  MoveL 3296 to (-321.69, 3.65, -16.53) mm, rotated rx -179.9 ry 0 rz -90 deg; joints [12.696, -89.548, 135.077, -162.211, 45.978, 167.852]
  MoveL 3297 to (-322.96, 3.57, -14.75) mm, rotated rx -179.9 ry 0 rz -90 deg; joints [12.649, -89.681, 135.215, -162.276, 45.973, 167.898]
  MoveL 3298 to (-323.52, 3.49, -12.64) mm, rotated rx -179.9 ry 0 rz -90 deg; joints [12.644, -89.825, 135.365, -162.283, 45.976, 167.904]
  MoveL 3299 to (-323.29, 3.42, -10.47) mm, rotated rx -179.9 ry 0 rz -90 deg; joints [12.684, -89.963, 135.506, -162.231, 45.988, 167.869]
  MoveL 3300 to (-322.29, 3.34, -8.52) mm, rotated rx -179.9 ry 0 rz -90 deg; joints [12.762, -90.074, 135.62, -162.126, 46.008, 167.798]
  MoveL 3301 to (-320.67, 3.26, -7.05) mm, rotated rx -179.9 ry 0 rz -90 deg; joints [12.868, -90.144, 135.694, -161.983, 46.035, 167.701]
  MoveL 3302 to (-318.64, 3.19, -6.26) mm, rotated rx -179.9 ry 0 rz -90 deg; joints [12.989, -90.162, 135.717, -161.82, 46.066, 167.592]
  MoveL 3303 to (-316.45, 3.11, -6.24) mm, rotated rx -179.9 ry 0 rz -90 deg; joints [13.109, -90.127, 135.687, -161.661, 46.097, 167.484]
  MoveL 3304 to (-314.4, 3.03, -7.01) mm, rotated rx -179.9 ry 0 rz -90 deg; joints [13.21, -90.041, 135.609, -161.525, 46.126, 167.394]
  MoveL 3305 to (-312.76, 2.96, -8.46) mm, rotated rx -179.9 ry 0 rz -90 deg; joints [13.28, -89.916, 135.492, -161.433, 46.15, 167.332]
  MoveL 3306 to (-311.74, 2.88, -10.39) mm, rotated rx -179.9 ry 0 rz -90 deg; joints [13.311, -89.769, 135.353, -161.394, 46.164, 167.308]
  MoveL 3307 to (-311.48, 2.8, -12.56) mm, rotated rx -179.9 ry 0 rz -90 deg; joints [13.297, -89.617, 135.21, -161.416, 46.169, 167.325]
  MoveL 3308 to (-312.01, 2.73, -14.68) mm, rotated rx -179.9 ry 0 rz -90 deg; joints [13.241, -89.482, 135.083, -161.493, 46.165, 167.38]
  MoveL 3309 to (-313.26, 2.65, -16.48) mm, rotated rx -179.9 ry 0 rz -90 deg; joints [13.151, -89.379, 134.988, -161.618, 46.152, 167.466]
  MoveL 3310 to (-315.07, 2.57, -17.71) mm, rotated rx -179.9 ry 0 rz -90 deg; joints [13.038, -89.322, 134.939, -161.773, 46.135, 167.573]
  MoveL 3311 to (-317.2, 2.5, -18.21) mm, rotated rx -179.9 ry 0 rz -90 deg; joints [12.918, -89.317, 134.941, -161.938, 46.116, 167.688]
  MoveL 3312 to (-319.37, 2.42, -17.92) mm, rotated rx -179.9 ry 0 rz -90 deg; joints [12.804, -89.364, 134.996, -162.094, 46.099, 167.796]
  MoveL 3313 to (-321.29, 2.34, -16.88) mm, rotated rx -179.9 ry 0 rz -90 deg; joints [12.714, -89.458, 135.097, -162.219, 46.086, 167.883]
  MoveL 3314 to (-322.71, 2.27, -15.22) mm, rotated rx -179.9 ry 0 rz -90 deg; joints [12.657, -89.585, 135.23, -162.298, 46.079, 167.937]
  MoveL 3315 to (-323.46, 2.19, -13.17) mm, rotated rx -179.9 ry 0 rz -90 deg; joints [12.642, -89.728, 135.378, -162.319, 46.081, 167.953]
  MoveL 3316 to (-323.42, 2.11, -10.98) mm, rotated rx -179.9 ry 0 rz -90 deg; joints [12.671, -89.869, 135.523, -162.281, 46.091, 167.928]
  MoveL 3317 to (-322.6, 2.04, -8.95) mm, rotated rx -179.9 ry 0 rz -90 deg; joints [12.741, -89.988, 135.646, -162.188, 46.109, 167.866]
  MoveL 3318 to (-321.11, 1.96, -7.35) mm, rotated rx -179.9 ry 0 rz -90 deg; joints [12.841, -90.069, 135.73, -162.052, 46.135, 167.774]
  MoveL 3319 to (-319.15, 1.88, -6.38) mm, rotated rx -179.9 ry 0 rz -90 deg; joints [12.96, -90.1, 135.766, -161.893, 46.165, 167.666]
  MoveL 3320 to (-316.98, 1.81, -6.18) mm, rotated rx -179.9 ry 0 rz -90 deg; joints [13.081, -90.077, 135.749, -161.731, 46.196, 167.557]
  MoveL 3321 to (-314.87, 1.73, -6.76) mm, rotated rx -179.9 ry 0 rz -90 deg; joints [13.188, -90.003, 135.681, -161.588, 46.226, 167.462]
  MoveL 3322 to (-313.11, 1.65, -8.05) mm, rotated rx -179.9 ry 0 rz -90 deg; joints [13.267, -89.886, 135.572, -161.484, 46.251, 167.393]
  MoveL 3323 to (-311.92, 1.57, -9.89) mm, rotated rx -179.9 ry 0 rz -90 deg; joints [13.308, -89.743, 135.437, -161.432, 46.268, 167.359]
  MoveL 3324 to (-311.47, 1.5, -12.03) mm, rotated rx -179.9 ry 0 rz -90 deg; joints [13.305, -89.591, 135.293, -161.438, 46.275, 167.366]
  MoveL 3325 to (-311.81, 1.42, -14.19) mm, rotated rx -179.9 ry 0 rz -90 deg; joints [13.259, -89.45, 135.16, -161.503, 46.272, 167.412]
  MoveL 3326 to (-312.9, 1.34, -16.09) mm, rotated rx -179.9 ry 0 rz -90 deg; joints [13.176, -89.338, 135.056, -161.617, 46.261, 167.491]
  MoveL 3327 to (-314.6, 1.27, -17.47) mm, rotated rx -179.9 ry 0 rz -90 deg; joints [13.067, -89.269, 134.995, -161.766, 46.245, 167.594]
  MoveL 3328 to (-316.67, 1.19, -18.16) mm, rotated rx -179.9 ry 0 rz -90 deg; joints [12.947, -89.251, 134.985, -161.931, 46.226, 167.708]
  MoveL 3329 to (-318.86, 1.11, -18.06) mm, rotated rx -179.9 ry 0 rz -90 deg; joints [12.831, -89.286, 135.028, -162.09, 46.208, 167.818]
  MoveL 3330 to (-320.86, 1.04, -17.2) mm, rotated rx -179.9 ry 0 rz -90 deg; joints [12.733, -89.369, 135.118, -162.224, 46.194, 167.911]
  MoveL 3331 to (-322.43, 0.96, -15.67) mm, rotated rx -179.9 ry 0 rz -90 deg; joints [12.667, -89.49, 135.244, -162.315, 46.187, 167.974]
  MoveL 3332 to (-323.35, 0.88, -13.69) mm, rotated rx -179.9 ry 0 rz -90 deg; joints [12.642, -89.631, 135.391, -162.351, 46.186, 168]
  MoveL 3333 to (-323.5, 0.81, -11.5) mm, rotated rx -179.9 ry 0 rz -90 deg; joints [12.661, -89.774, 135.539, -162.328, 46.195, 167.985]
  MoveL 3334 to (-322.86, 0.73, -9.41) mm, rotated rx -179.9 ry 0 rz -90 deg; joints [12.721, -89.9, 135.668, -162.247, 46.211, 167.931]
  MoveL 3335 to (-321.52, 0.65, -7.69) mm, rotated rx -179.9 ry 0 rz -90 deg; joints [12.815, -89.991, 135.763, -162.12, 46.235, 167.845]
  MoveL 3336 to (-319.65, 0.58, -6.55) mm, rotated rx -179.9 ry 0 rz -90 deg; joints [12.931, -90.035, 135.812, -161.965, 46.264, 167.741]
  MoveL 3337 to (-317.5, 0.5, -6.15) mm, rotated rx -179.9 ry 0 rz -90 deg; joints [13.053, -90.025, 135.807, -161.802, 46.295, 167.631]
  MoveL 3338 to (-317.17, 0.5, -6.15) mm, rotated rx -179.9 ry 0 rz -90 deg; joints [13.071, -90.02, 135.802, -161.777, 46.299, 167.614]
  MoveC 3339 to (-315.68, 0.5, -6.77) mm, rotated rx -179.9 ry 0 rz -90 deg; joints [13.145, -89.956, 135.739, -161.678, 46.316, 167.547] to (-315.06, 0.5, -8.27) mm, rotated rx -179.9 ry 0 rz -90 deg; joints [13.159, -89.848, 135.632, -161.659, 46.32, 167.535]
  MoveL 3340 to (-315.06, 0.5, -8.27) mm, rotated rx -179.9 ry 0 rz -90 deg; joints [13.159, -89.848, 135.632, -161.659, 46.32, 167.535]
  MoveL 3341 to (-315.06, 0.5, -303.97) mm, rotated rx -179.9 ry 0 rz -90 deg; joints [10.211, -71.759, 114.391, -164.852, 42.693, 169.127]
  MoveC 3342 to (-315.68, 0.5, -305.46) mm, rotated rx -179.9 ry 0 rz -90 deg; joints [10.173, -71.679, 114.282, -164.899, 42.658, 169.156] to (-317.17, 0.5, -306.08) mm, rotated rx -179.9 ry 0 rz -90 deg; joints [10.104, -71.658, 114.254, -164.997, 42.639, 169.225]
  MoveL 3343 to (-317.17, 0.5, -306.08) mm, rotated rx -179.9 ry 0 rz -90 deg; joints [10.104, -71.658, 114.254, -164.997, 42.639, 169.225]
  MoveL 3344 to (-317.84, 0.5, -306.08) mm, rotated rx -179.9 ry 0 rz -90 deg; joints [10.076, -71.665, 114.264, -165.039, 42.636, 169.256]
  MoveC 3345 to (-319.33, 0.5, -305.46) mm, rotated rx -179.9 ry 0 rz -90 deg; joints [10.016, -71.716, 114.334, -165.13, 42.643, 169.326] to (-319.95, 0.5, -303.97) mm, rotated rx -179.9 ry 0 rz -90 deg; joints [10.001, -71.809, 114.461, -165.161, 42.673, 169.354]
  MoveL 3346 to (-319.95, 0.5, -303.97) mm, rotated rx -179.9 ry 0 rz -90 deg; joints [10.001, -71.809, 114.461, -165.161, 42.673, 169.354]
  MoveL 3347 to (-319.95, 0.5, -8.27) mm, rotated rx -179.9 ry 0 rz -90 deg; joints [12.894, -89.922, 135.707, -162.018, 46.264, 167.779]
  MoveC 3348 to (-319.33, 0.5, -6.77) mm, rotated rx -179.9 ry 0 rz -90 deg; joints [12.946, -90.012, 135.795, -161.947, 46.273, 167.73] to (-317.84, 0.5, -6.15) mm, rotated rx -179.9 ry 0 rz -90 deg; joints [13.035, -90.03, 135.812, -161.826, 46.292, 167.648]
  MoveL 3349 to (-317.84, 0.5, -6.15) mm, rotated rx -179.9 ry 0 rz -90 deg; joints [13.035, -90.03, 135.812, -161.826, 46.292, 167.648]
  MoveL 3350 to (-317.5, 0.5, -6.15) mm, rotated rx -179.9 ry 0 rz -90 deg; joints [13.053, -90.025, 135.807, -161.802, 46.295, 167.631]
  MoveC 3351 to (-315.43, 0.5, -5.57) mm, rotated rx -179.9 ry 0 rz -90 deg; joints [13.174, -90.032, 135.813, -161.639, 46.32, 167.52] to (-313.95, 0.5, -4) mm, rotated rx -179.9 ry 0 rz -90 deg; joints [13.275, -90.114, 135.892, -161.502, 46.34, 167.427]
  MoveL 3352 to (-313.95, 0.5, -4) mm, rotated rx -179.9 ry 0 rz -90 deg; joints [13.275, -90.114, 135.892, -161.502, 46.34, 167.427]
  MoveC 3353 to (-311.54, 0.5, -2.91) mm, rotated rx -179.9 ry 0 rz -90 deg; joints [13.42, -90.149, 135.924, -161.306, 46.37, 167.293] to (-309.91, 0.5, -4.99) mm, rotated rx -179.9 ry 0 rz -90 deg; joints [13.481, -89.985, 135.763, -161.224, 46.386, 167.238]
  MoveL 3354 to (-309.91, 0.5, -4.99) mm, rotated rx -179.9 ry 0 rz -90 deg; joints [13.481, -89.985, 135.763, -161.224, 46.386, 167.238]
  MoveL 3355 to (-309.91, 0.5, -311.23) mm, rotated rx -179.9 ry 0 rz -90 deg; joints [10.374, -71.283, 113.739, -164.566, 42.556, 168.888]
  MoveL 3356 to (-325.1, 0.5, -311.23) mm, rotated rx -179.9 ry 0 rz -90 deg; joints [9.727, -71.437, 113.959, -165.524, 42.495, 169.594]
  MoveL 3357 to (-325.1, 0.5, -1) mm, rotated rx -179.9 ry 0 rz -90 deg; joints [12.703, -90.482, 136.257, -162.273, 46.213, 167.95]
  MoveL 3358 to (-309.91, 0.5, -1) mm, rotated rx -179.9 ry 0 rz -90 deg; joints [13.534, -90.25, 136.022, -161.151, 46.392, 167.188]
  MoveL 3359 to (-309.91, 0.5, -4.99) mm, rotated rx -179.9 ry 0 rz -90 deg; joints [13.481, -89.985, 135.763, -161.224, 46.386, 167.238]
  MoveL 3360 to (-309.93, 0.52, -5.21) mm, rotated rx -179.9 ry 0 rz -90 deg; joints [13.477, -89.972, 135.749, -161.229, 46.384, 167.241]
  MoveL 3361 to (-309.98, 0.58, -5.42) mm, rotated rx -179.9 ry 0 rz -90 deg; joints [13.472, -89.962, 135.734, -161.235, 46.379, 167.244]
  MoveL 3362 to (-310.06, 0.67, -5.6) mm, rotated rx -179.9 ry 0 rz -90 deg; joints [13.465, -89.955, 135.72, -161.242, 46.37, 167.247]
  MoveL 3363 to (-310.16, 0.8, -5.75) mm, rotated rx -179.9 ry 0 rz -90 deg; joints [13.457, -89.953, 135.707, -161.249, 46.358, 167.249]
  MoveL 3364 to (-310.26, 0.95, -5.87) mm, rotated rx -179.9 ry 0 rz -90 deg; joints [13.45, -89.954, 135.695, -161.254, 46.344, 167.25]
  MoveL 3365 to (-310.36, 1.13, -5.96) mm, rotated rx -179.9 ry 0 rz -90 deg; joints [13.444, -89.958, 135.684, -161.258, 46.328, 167.249]
  MoveL 3366 to (-310.43, 1.34, -6.02) mm, rotated rx -179.9 ry 0 rz -90 deg; joints [13.439, -89.965, 135.674, -161.259, 46.311, 167.246]
  MoveL 3367 to (-310.48, 1.55, -6.05) mm, rotated rx -179.9 ry 0 rz -90 deg; joints [13.436, -89.974, 135.665, -161.258, 46.293, 167.241]
  MoveL 3368 to (-310.49, 1.77, -6.06) mm, rotated rx -179.9 ry 0 rz -90 deg; joints [13.435, -89.984, 135.656, -161.254, 46.276, 167.233]
  Set speed (1000.0 mm/s)
  MoveL 3369 to (-310.49, 185.53, -6.06) mm, rotated rx -179.9 ry 0 rz -90 deg; joints [13.36, -96.669, 127.503, -154.519, 32.472, 158.531]
  Print: /'Contour3'
  Call SetTool(1)
  Set speed (1000.0 mm/s)
  MoveL 3370 to (-315.03, 25.52, 4.01) mm, rotated rx -179.9 ry 0 rz -90 deg; joints [13.309, -91.824, 135.461, -160.771, 44.323, 166.421]
  MoveL 3371 to (-315.03, 11.79, 4.01) mm, rotated rx -179.9 ry 0 rz -90 deg; joints [13.315, -91.197, 135.998, -161.144, 45.423, 166.953]
  Set speed (100.0 mm/s)
  MoveL 3372 to (-315.03, 4.8, 4.01) mm, rotated rx -179.9 ry 0 rz -90 deg; joints [13.318, -90.869, 136.265, -161.327, 45.987, 167.218]
  MoveL 3373 to (-314.68, 3.9, 3.89) mm, rotated rx -179.9 ry 0 rz -90 deg; joints [13.336, -90.813, 136.286, -161.326, 46.064, 167.236]
  MoveL 3374 to (-313.82, 3.52, 3.62) mm, rotated rx -179.9 ry 0 rz -90 deg; joints [13.38, -90.764, 136.269, -161.277, 46.105, 167.21]
  MoveL 3375 to (-309.98, 3.52, 2.4) mm, rotated rx -179.9 ry 0 rz -90 deg; joints [13.574, -90.622, 136.13, -161.015, 46.151, 167.032]
  MoveC 3376 to (-309.23, 3.53, 1.78) mm, rotated rx -179.9 ry 0 rz -90 deg; joints [13.606, -90.568, 136.077, -160.972, 46.16, 167.003] to (-309.15, 3.53, 0.81) mm, rotated rx -179.9 ry 0 rz -90 deg; joints [13.598, -90.502, 136.014, -160.984, 46.16, 167.012]
  MoveL 3377 to (-309.15, 3.52, 0.81) mm, rotated rx -179.9 ry 0 rz -90 deg; joints [13.598, -90.502, 136.014, -160.984, 46.16, 167.012]
  MoveL 3378 to (-309.24, 3.53, 0.47) mm, rotated rx -179.9 ry 0 rz -90 deg; joints [13.588, -90.481, 135.993, -160.997, 46.159, 167.021]
  MoveL 3379 to (-309.31, 3.52, 0.13) mm, rotated rx -179.9 ry 0 rz -90 deg; joints [13.58, -90.46, 135.972, -161.009, 46.157, 167.029]
  MoveL 3380 to (-309.38, 3.52, -0.32) mm, rotated rx -179.9 ry 0 rz -90 deg; joints [13.57, -90.431, 135.944, -161.022, 46.156, 167.038]
  MoveL 3381 to (-309.41, 3.52, -0.77) mm, rotated rx -179.9 ry 0 rz -90 deg; joints [13.563, -90.401, 135.916, -161.032, 46.155, 167.045]
  MoveL 3382 to (-309.41, 3.52, -1.67) mm, rotated rx -179.9 ry 0 rz -90 deg; joints [13.551, -90.342, 135.858, -161.049, 46.154, 167.057]
  MoveL 3383 to (-309.41, 3.53, -310.57) mm, rotated rx -179.9 ry 0 rz -90 deg; joints [10.399, -71.426, 113.69, -164.473, 42.376, 168.785]
  MoveL 3384 to (-309.41, 3.52, -311.47) mm, rotated rx -179.9 ry 0 rz -90 deg; joints [10.392, -71.373, 113.619, -164.478, 42.356, 168.785]
  MoveL 3385 to (-309.38, 3.52, -311.92) mm, rotated rx -179.9 ry 0 rz -90 deg; joints [10.39, -71.347, 113.583, -164.478, 42.347, 168.783]
  MoveL 3386 to (-309.31, 3.52, -312.37) mm, rotated rx -179.9 ry 0 rz -90 deg; joints [10.389, -71.32, 113.546, -164.476, 42.337, 168.78]
  MoveL 3387 to (-309.24, 3.52, -312.7) mm, rotated rx -179.9 ry 0 rz -90 deg; joints [10.39, -71.299, 113.518, -164.474, 42.33, 168.777]
  MoveL 3388 to (-309.15, 3.53, -313.04) mm, rotated rx -179.9 ry 0 rz -90 deg; joints [10.391, -71.279, 113.49, -164.47, 42.323, 168.773]
  MoveL 3389 to (-309.08, 3.53, -313.26) mm, rotated rx -179.9 ry 0 rz -90 deg; joints [10.392, -71.265, 113.471, -164.466, 42.318, 168.769]
  MoveL 3390 to (-308.91, 3.52, -313.71) mm, rotated rx -179.9 ry 0 rz -90 deg; joints [10.396, -71.237, 113.433, -164.458, 42.309, 168.761]
  MoveL 3391 to (-308.7, 3.52, -314.16) mm, rotated rx -179.9 ry 0 rz -90 deg; joints [10.401, -71.209, 113.394, -164.447, 42.3, 168.751]
  MoveL 3392 to (-308.49, 3.53, -314.53) mm, rotated rx -179.9 ry 0 rz -90 deg; joints [10.407, -71.185, 113.362, -164.436, 42.293, 168.742]
  MoveL 3393 to (-308.25, 3.53, -314.9) mm, rotated rx -179.9 ry 0 rz -90 deg; joints [10.414, -71.161, 113.329, -164.423, 42.286, 168.73]
  MoveL 3394 to (-308.13, 3.52, -315.06) mm, rotated rx -179.9 ry 0 rz -90 deg; joints [10.418, -71.15, 113.314, -164.416, 42.283, 168.725]
  MoveL 3395 to (-307.96, 3.53, -315.27) mm, rotated rx -179.9 ry 0 rz -90 deg; joints [10.424, -71.136, 113.295, -164.406, 42.278, 168.717]
  MoveL 3396 to (-307.78, 3.53, -315.49) mm, rotated rx -179.9 ry 0 rz -90 deg; joints [10.43, -71.122, 113.275, -164.396, 42.274, 168.708]
  MoveL 3397 to (-307.57, 3.52, -315.7) mm, rotated rx -179.9 ry 0 rz -90 deg; joints [10.437, -71.107, 113.255, -164.384, 42.271, 168.699]
  MoveL 3398 to (-307.35, 3.53, -315.92) mm, rotated rx -179.9 ry 0 rz -90 deg; joints [10.444, -71.092, 113.234, -164.371, 42.267, 168.688]
  MoveL 3399 to (-307.31, 3.52, -315.96) mm, rotated rx -179.9 ry 0 rz -90 deg; joints [10.446, -71.089, 113.23, -164.369, 42.266, 168.686]
  MoveL 3400 to (-306.88, 3.52, -316.31) mm, rotated rx -179.9 ry 0 rz -90 deg; joints [10.461, -71.064, 113.196, -164.343, 42.26, 168.666]
  MoveL 3401 to (-306.45, 3.53, -316.6) mm, rotated rx -179.9 ry 0 rz -90 deg; joints [10.477, -71.043, 113.166, -164.318, 42.255, 168.646]
  MoveL 3402 to (-306.02, 3.53, -316.86) mm, rotated rx -179.9 ry 0 rz -90 deg; joints [10.493, -71.023, 113.139, -164.292, 42.251, 168.626]
  MoveL 3403 to (-305.55, 3.53, -317.08) mm, rotated rx -179.9 ry 0 rz -90 deg; joints [10.511, -71.006, 113.115, -164.264, 42.249, 168.604]
  MoveL 3404 to (-305.1, 3.52, -317.25) mm, rotated rx -179.9 ry 0 rz -90 deg; joints [10.529, -70.991, 113.094, -164.237, 42.247, 168.583]
  MoveL 3405 to (-304.66, 3.53, -317.38) mm, rotated rx -179.9 ry 0 rz -90 deg; joints [10.547, -70.978, 113.077, -164.209, 42.245, 168.562]
  MoveL 3406 to (-304.21, 3.52, -317.48) mm, rotated rx -179.9 ry 0 rz -90 deg; joints [10.565, -70.968, 113.062, -164.181, 42.245, 168.541]
  MoveL 3407 to (-303.76, 3.53, -317.55) mm, rotated rx -179.9 ry 0 rz -90 deg; joints [10.583, -70.959, 113.05, -164.153, 42.246, 168.52]
  MoveL 3408 to (-303.31, 3.52, -317.58) mm, rotated rx -179.9 ry 0 rz -90 deg; joints [10.602, -70.952, 113.04, -164.125, 42.247, 168.499]
  MoveL 3409 to (-302.86, 3.53, -317.59) mm, rotated rx -179.9 ry 0 rz -90 deg; joints [10.621, -70.947, 113.033, -164.097, 42.248, 168.478]
  MoveL 3410 to (315.44, 3.53, -317.59) mm, rotated rx -179.9 ry 0 rz -90 deg; joints [33.379, -56.906, 91.665, -130.07, 45.953, 141.252]
  MoveL 3411 to (315.89, 3.53, -317.58) mm, rotated rx -179.9 ry 0 rz -90 deg; joints [33.393, -56.891, 91.641, -130.048, 45.956, 141.232]
  MoveL 3412 to (316.34, 3.52, -317.54) mm, rotated rx -179.9 ry 0 rz -90 deg; joints [33.407, -56.878, 91.62, -130.026, 45.96, 141.213]
  MoveL 3413 to (316.79, 3.53, -317.47) mm, rotated rx -179.9 ry 0 rz -90 deg; joints [33.422, -56.866, 91.601, -130.004, 45.965, 141.194]
  MoveL 3414 to (317.24, 3.52, -317.36) mm, rotated rx -179.9 ry 0 rz -90 deg; joints [33.438, -56.856, 91.584, -129.983, 45.97, 141.175]
  MoveL 3415 to (317.69, 3.53, -317.23) mm, rotated rx -179.9 ry 0 rz -90 deg; joints [33.454, -56.848, 91.571, -129.961, 45.977, 141.158]
  MoveL 3416 to (318.14, 3.52, -317.05) mm, rotated rx -179.9 ry 0 rz -90 deg; joints [33.472, -56.842, 91.561, -129.939, 45.986, 141.141]
  MoveL 3417 to (318.54, 3.52, -316.86) mm, rotated rx -179.9 ry 0 rz -90 deg; joints [33.488, -56.838, 91.555, -129.92, 45.994, 141.126]
  MoveL 3418 to (318.78, 3.52, -316.72) mm, rotated rx -179.9 ry 0 rz -90 deg; joints [33.498, -56.837, 91.552, -129.908, 46, 141.117]
  MoveL 3419 to (319.03, 3.53, -316.56) mm, rotated rx -179.9 ry 0 rz -90 deg; joints [33.509, -56.836, 91.551, -129.896, 46.006, 141.109]
  MoveL 3420 to (319.43, 3.52, -316.28) mm, rotated rx -179.9 ry 0 rz -90 deg; joints [33.526, -56.837, 91.552, -129.877, 46.018, 141.096]
  MoveL 3421 to (319.83, 3.52, -315.96) mm, rotated rx -179.9 ry 0 rz -90 deg; joints [33.545, -56.841, 91.557, -129.859, 46.03, 141.084]
  MoveL 3422 to (319.93, 3.53, -315.86) mm, rotated rx -179.9 ry 0 rz -90 deg; joints [33.55, -56.842, 91.56, -129.853, 46.034, 141.081]
  MoveL 3423 to (320.14, 3.52, -315.66) mm, rotated rx -179.9 ry 0 rz -90 deg; joints [33.56, -56.846, 91.565, -129.844, 46.042, 141.076]
  MoveL 3424 to (320.32, 3.52, -315.46) mm, rotated rx -179.9 ry 0 rz -90 deg; joints [33.57, -56.85, 91.571, -129.835, 46.049, 141.071]
  MoveL 3425 to (320.65, 3.53, -315.06) mm, rotated rx -179.9 ry 0 rz -90 deg; joints [33.588, -56.859, 91.586, -129.82, 46.064, 141.063]
  MoveL 3426 to (320.83, 3.52, -314.8) mm, rotated rx -179.9 ry 0 rz -90 deg; joints [33.599, -56.866, 91.597, -129.811, 46.073, 141.06]
  MoveL 3427 to (321.04, 3.52, -314.48) mm, rotated rx -179.9 ry 0 rz -90 deg; joints [33.612, -56.876, 91.612, -129.801, 46.085, 141.056]
  MoveL 3428 to (321.22, 3.52, -314.16) mm, rotated rx -179.9 ry 0 rz -90 deg; joints [33.623, -56.887, 91.629, -129.793, 46.096, 141.054]
  MoveL 3429 to (321.43, 3.53, -313.71) mm, rotated rx -179.9 ry 0 rz -90 deg; joints [33.639, -56.903, 91.654, -129.783, 46.112, 141.053]
  MoveL 3430 to (321.6, 3.53, -313.26) mm, rotated rx -179.9 ry 0 rz -90 deg; joints [33.653, -56.92, 91.682, -129.775, 46.127, 141.053]
  MoveL 3431 to (321.73, 3.53, -312.81) mm, rotated rx -179.9 ry 0 rz -90 deg; joints [33.666, -56.939, 91.711, -129.769, 46.143, 141.055]
  MoveL 3432 to (321.83, 3.52, -312.37) mm, rotated rx -179.9 ry 0 rz -90 deg; joints [33.678, -56.959, 91.743, -129.765, 46.158, 141.059]
  MoveL 3433 to (321.89, 3.52, -311.92) mm, rotated rx -179.9 ry 0 rz -90 deg; joints [33.69, -56.98, 91.776, -129.762, 46.173, 141.064]
  MoveL 3434 to (321.93, 3.52, -311.47) mm, rotated rx -179.9 ry 0 rz -90 deg; joints [33.7, -57.002, 91.811, -129.761, 46.187, 141.07]
  MoveL 3435 to (321.93, 3.52, -310.57) mm, rotated rx -179.9 ry 0 rz -90 deg; joints [33.718, -57.049, 91.885, -129.761, 46.216, 141.086]
  MoveL 3436 to (321.93, 3.52, -1.67) mm, rotated rx -179.9 ry 0 rz -90 deg; joints [41.183, -71.832, 113.655, -126.643, 55.135, 143.485]
  MoveL 3437 to (321.93, 3.52, -0.77) mm, rotated rx -179.9 ry 0 rz -90 deg; joints [41.209, -71.873, 113.709, -126.626, 55.158, 143.485]
  MoveL 3438 to (321.89, 3.52, -0.32) mm, rotated rx -179.9 ry 0 rz -90 deg; joints [41.221, -71.894, 113.738, -126.619, 55.17, 143.486]
  MoveL 3439 to (321.83, 3.53, 0.13) mm, rotated rx -179.9 ry 0 rz -90 deg; joints [41.231, -71.917, 113.769, -126.613, 55.181, 143.487]
  MoveL 3440 to (321.73, 3.52, 0.58) mm, rotated rx -179.9 ry 0 rz -90 deg; joints [41.241, -71.941, 113.801, -126.608, 55.192, 143.49]
  MoveL 3441 to (321.6, 3.53, 1.03) mm, rotated rx -179.9 ry 0 rz -90 deg; joints [41.25, -71.966, 113.835, -126.605, 55.202, 143.494]
  MoveL 3442 to (321.43, 3.53, 1.48) mm, rotated rx -179.9 ry 0 rz -90 deg; joints [41.257, -71.993, 113.871, -126.603, 55.212, 143.5]
  MoveL 3443 to (321.22, 3.52, 1.93) mm, rotated rx -179.9 ry 0 rz -90 deg; joints [41.263, -72.021, 113.91, -126.603, 55.221, 143.506]
  MoveL 3444 to (321.04, 3.53, 2.25) mm, rotated rx -179.9 ry 0 rz -90 deg; joints [41.266, -72.042, 113.938, -126.603, 55.228, 143.512]
  MoveL 3445 to (320.83, 3.52, 2.57) mm, rotated rx -179.9 ry 0 rz -90 deg; joints [41.269, -72.065, 113.969, -126.605, 55.234, 143.518]
  MoveL 3446 to (320.65, 3.53, 2.82) mm, rotated rx -179.9 ry 0 rz -90 deg; joints [41.27, -72.083, 113.994, -126.608, 55.239, 143.524]
  MoveL 3447 to (320.32, 3.52, 3.22) mm, rotated rx -179.9 ry 0 rz -90 deg; joints [41.271, -72.114, 114.035, -126.613, 55.246, 143.534]
  MoveL 3448 to (320.14, 3.52, 3.42) mm, rotated rx -179.9 ry 0 rz -90 deg; joints [41.271, -72.13, 114.057, -126.617, 55.249, 143.54]
  MoveL 3449 to (319.93, 3.52, 3.62) mm, rotated rx -179.9 ry 0 rz -90 deg; joints [41.27, -72.147, 114.08, -126.621, 55.252, 143.546]
  MoveL 3450 to (319.83, 3.53, 3.72) mm, rotated rx -179.9 ry 0 rz -90 deg; joints [41.269, -72.156, 114.092, -126.623, 55.254, 143.55]
  MoveL 3451 to (319.43, 3.53, 4.05) mm, rotated rx -179.9 ry 0 rz -90 deg; joints [41.266, -72.186, 114.133, -126.633, 55.258, 143.562]
  MoveL 3452 to (319.03, 3.52, 4.33) mm, rotated rx -179.9 ry 0 rz -90 deg; joints [41.261, -72.214, 114.171, -126.643, 55.261, 143.574]
  MoveL 3453 to (318.79, 3.53, 4.48) mm, rotated rx -179.9 ry 0 rz -90 deg; joints [41.257, -72.23, 114.193, -126.65, 55.262, 143.582]
  MoveL 3454 to (318.54, 3.53, 4.62) mm, rotated rx -179.9 ry 0 rz -90 deg; joints [41.253, -72.246, 114.215, -126.657, 55.263, 143.59]
  MoveL 3455 to (318.14, 3.52, 4.81) mm, rotated rx -179.9 ry 0 rz -90 deg; joints [41.245, -72.27, 114.248, -126.669, 55.264, 143.603]
  MoveL 3456 to (317.69, 3.52, 4.99) mm, rotated rx -179.9 ry 0 rz -90 deg; joints [41.236, -72.296, 114.282, -126.684, 55.264, 143.617]
  MoveL 3457 to (317.24, 3.52, 5.13) mm, rotated rx -179.9 ry 0 rz -90 deg; joints [41.225, -72.319, 114.315, -126.699, 55.263, 143.631]
  MoveL 3458 to (316.79, 3.52, 5.23) mm, rotated rx -179.9 ry 0 rz -90 deg; joints [41.213, -72.342, 114.345, -126.715, 55.26, 143.645]
  MoveL 3459 to (316.34, 3.52, 5.3) mm, rotated rx -179.9 ry 0 rz -90 deg; joints [41.201, -72.362, 114.373, -126.732, 55.257, 143.659]
  MoveL 3460 to (315.89, 3.53, 5.34) mm, rotated rx -179.9 ry 0 rz -90 deg; joints [41.187, -72.381, 114.399, -126.749, 55.254, 143.674]
  MoveL 3461 to (315.44, 3.52, 5.35) mm, rotated rx -179.9 ry 0 rz -90 deg; joints [41.172, -72.399, 114.424, -126.767, 55.249, 143.688]
  MoveL 3462 to (-302.86, 3.52, 5.35) mm, rotated rx -179.9 ry 0 rz -90 deg; joints [14.002, -90.704, 136.204, -160.435, 46.243, 166.636]
  MoveL 3463 to (-303.31, 3.52, 5.35) mm, rotated rx -179.9 ry 0 rz -90 deg; joints [13.978, -90.711, 136.211, -160.468, 46.238, 166.659]
  MoveL 3464 to (-303.76, 3.52, 5.31) mm, rotated rx -179.9 ry 0 rz -90 deg; joints [13.953, -90.716, 136.216, -160.502, 46.232, 166.682]
  MoveL 3465 to (-304.21, 3.52, 5.25) mm, rotated rx -179.9 ry 0 rz -90 deg; joints [13.927, -90.719, 136.22, -160.536, 46.226, 166.705]
  MoveL 3466 to (-304.66, 3.53, 5.15) mm, rotated rx -179.9 ry 0 rz -90 deg; joints [13.901, -90.72, 136.22, -160.571, 46.22, 166.729]
  MoveL 3467 to (-305.1, 3.53, 5.01) mm, rotated rx -179.9 ry 0 rz -90 deg; joints [13.875, -90.718, 136.219, -160.607, 46.215, 166.753]
  MoveL 3468 to (-305.55, 3.53, 4.84) mm, rotated rx -179.9 ry 0 rz -90 deg; joints [13.848, -90.714, 136.215, -160.643, 46.209, 166.778]
  MoveL 3469 to (-306.02, 3.53, 4.62) mm, rotated rx -179.9 ry 0 rz -90 deg; joints [13.82, -90.706, 136.209, -160.682, 46.203, 166.804]
  MoveL 3470 to (-306.45, 3.52, 4.37) mm, rotated rx -179.9 ry 0 rz -90 deg; joints [13.793, -90.697, 136.2, -160.719, 46.197, 166.829]
  MoveL 3471 to (-306.88, 3.53, 4.07) mm, rotated rx -179.9 ry 0 rz -90 deg; joints [13.765, -90.684, 136.188, -160.756, 46.191, 166.855]
  MoveL 3472 to (-307.31, 3.52, 3.72) mm, rotated rx -179.9 ry 0 rz -90 deg; joints [13.737, -90.667, 136.172, -160.794, 46.186, 166.881]
  MoveL 3473 to (-307.35, 3.53, 3.68) mm, rotated rx -179.9 ry 0 rz -90 deg; joints [13.734, -90.665, 136.17, -160.798, 46.185, 166.884]
  MoveL 3474 to (-307.57, 3.53, 3.47) mm, rotated rx -179.9 ry 0 rz -90 deg; joints [13.719, -90.655, 136.16, -160.818, 46.182, 166.898]
  MoveL 3475 to (-307.78, 3.53, 3.25) mm, rotated rx -179.9 ry 0 rz -90 deg; joints [13.705, -90.644, 136.149, -160.837, 46.179, 166.911]
  MoveL 3476 to (-307.96, 3.53, 3.04) mm, rotated rx -179.9 ry 0 rz -90 deg; joints [13.692, -90.632, 136.138, -160.855, 46.177, 166.923]
  MoveL 3477 to (-308.13, 3.53, 2.82) mm, rotated rx -179.9 ry 0 rz -90 deg; joints [13.68, -90.621, 136.127, -160.871, 46.175, 166.934]
  MoveL 3478 to (-308.25, 3.53, 2.66) mm, rotated rx -179.9 ry 0 rz -90 deg; joints [13.672, -90.612, 136.119, -160.883, 46.173, 166.942]
  MoveL 3479 to (-308.49, 3.52, 2.29) mm, rotated rx -179.9 ry 0 rz -90 deg; joints [13.653, -90.591, 136.099, -160.908, 46.17, 166.959]
  MoveL 3480 to (-308.7, 3.52, 1.93) mm, rotated rx -179.9 ry 0 rz -90 deg; joints [13.637, -90.57, 136.078, -160.93, 46.167, 166.974]
  MoveL 3481 to (-308.91, 3.52, 1.48) mm, rotated rx -179.9 ry 0 rz -90 deg; joints [13.62, -90.543, 136.053, -160.954, 46.164, 166.991]
  MoveL 3482 to (-309.08, 3.53, 1.03) mm, rotated rx -179.9 ry 0 rz -90 deg; joints [13.605, -90.516, 136.027, -160.975, 46.161, 167.005]
  MoveL 3483 to (-309.15, 3.52, 0.81) mm, rotated rx -179.9 ry 0 rz -90 deg; joints [13.598, -90.502, 136.014, -160.984, 46.16, 167.012]
  MoveC 3484 to (-309.77, 3.53, 0.07) mm, rotated rx -179.9 ry 0 rz -90 deg; joints [13.554, -90.463, 135.976, -161.044, 46.152, 167.053] to (-310.74, 3.52, -0.02) mm, rotated rx -179.9 ry 0 rz -90 deg; joints [13.5, -90.472, 135.986, -161.117, 46.14, 167.103]
  MoveL 3485 to (-310.74, 3.53, -0.02) mm, rotated rx -179.9 ry 0 rz -90 deg; joints [13.5, -90.472, 135.986, -161.117, 46.14, 167.103]
  MoveC 3486 to (-311.92, 3.53, -0.24) mm, rotated rx -179.9 ry 0 rz -90 deg; joints [13.433, -90.476, 135.99, -161.208, 46.125, 167.165] to (-312.39, 3.52, -1.34) mm, rotated rx -179.9 ry 0 rz -90 deg; joints [13.393, -90.41, 135.926, -161.263, 46.118, 167.203]
  MoveL 3487 to (-312.39, 3.52, -1.34) mm, rotated rx -179.9 ry 0 rz -90 deg; joints [13.393, -90.41, 135.926, -161.263, 46.118, 167.203]
  MoveC 3488 to (-312.56, 3.53, -2.1) mm, rotated rx -179.9 ry 0 rz -90 deg; joints [13.373, -90.362, 135.88, -161.289, 46.115, 167.221] to (-313.14, 3.53, -2.61) mm, rotated rx -179.9 ry 0 rz -90 deg; joints [13.335, -90.337, 135.856, -161.341, 46.108, 167.257]
  MoveL 3489 to (-313.14, 3.52, -2.61) mm, rotated rx -179.9 ry 0 rz -90 deg; joints [13.335, -90.337, 135.856, -161.341, 46.108, 167.257]
  MoveC 3490 to (-321.1, 3.53, 0.46) mm, rotated rx -179.9 ry 0 rz -90 deg; joints [12.94, -90.664, 136.178, -161.875, 46.015, 167.62] to (-318.03, 3.52, 8.42) mm, rotated rx -179.9 ry 0 rz -90 deg; joints [13.211, -91.152, 136.644, -161.501, 46.054, 167.359]
  MoveL 3491 to (-318.03, 3.52, 8.42) mm, rotated rx -179.9 ry 0 rz -90 deg; joints [13.211, -91.152, 136.644, -161.501, 46.054, 167.359]
  MoveC 3492 to (-310.52, 3.52, 6.18) mm, rotated rx -179.9 ry 0 rz -90 deg; joints [13.594, -90.883, 136.382, -160.985, 46.147, 167.009] to (-311.55, 3.52, -1.58) mm, rotated rx -179.9 ry 0 rz -90 deg; joints [13.435, -90.381, 135.897, -161.205, 46.128, 167.164]
  MoveL 3493 to (-311.55, 3.53, -1.58) mm, rotated rx -179.9 ry 0 rz -90 deg; joints [13.435, -90.381, 135.897, -161.205, 46.128, 167.164]
  MoveL 3494 to (-311.58, 3.52, -1.61) mm, rotated rx -179.9 ry 0 rz -90 deg; joints [13.433, -90.379, 135.896, -161.208, 46.128, 167.166]
  MoveL 3495 to (-313.45, 3.45, -2.74) mm, rotated rx -179.9 ry 0 rz -90 deg; joints [13.317, -90.33, 135.855, -161.368, 46.11, 167.277]
  MoveL 3496 to (-315.6, 3.37, -3.13) mm, rotated rx -179.9 ry 0 rz -90 deg; joints [13.195, -90.333, 135.866, -161.536, 46.09, 167.393]
  MoveL 3497 to (-317.75, 3.29, -2.73) mm, rotated rx -179.9 ry 0 rz -90 deg; joints [13.083, -90.389, 135.928, -161.689, 46.071, 167.499]
  MoveL 3498 to (-319.61, 3.22, -1.59) mm, rotated rx -179.9 ry 0 rz -90 deg; joints [12.996, -90.49, 136.034, -161.809, 46.056, 167.581]
  MoveL 3499 to (-320.94, 3.14, 0.13) mm, rotated rx -179.9 ry 0 rz -90 deg; joints [12.944, -90.622, 136.169, -161.879, 46.048, 167.63]
  MoveL 3500 to (-321.58, 3.06, 2.22) mm, rotated rx -179.9 ry 0 rz -90 deg; joints [12.936, -90.768, 136.316, -161.891, 46.048, 167.638]
  MoveL 3501 to (-321.43, 2.99, 4.4) mm, rotated rx -179.9 ry 0 rz -90 deg; joints [12.972, -90.908, 136.457, -161.842, 46.056, 167.605]
  MoveL 3502 to (-320.51, 2.91, 6.38) mm, rotated rx -179.9 ry 0 rz -90 deg; joints [13.048, -91.024, 136.574, -161.74, 46.074, 167.536]
  MoveL 3503 to (-318.96, 2.83, 7.91) mm, rotated rx -179.9 ry 0 rz -90 deg; joints [13.153, -91.099, 136.651, -161.597, 46.099, 167.439]
  MoveL 3504 to (-316.95, 2.76, 8.78) mm, rotated rx -179.9 ry 0 rz -90 deg; joints [13.275, -91.123, 136.679, -161.434, 46.13, 167.329]
  MoveL 3505 to (-314.77, 2.68, 8.88) mm, rotated rx -179.9 ry 0 rz -90 deg; joints [13.397, -91.092, 136.655, -161.272, 46.163, 167.22]
  MoveL 3506 to (-312.7, 2.61, 8.2) mm, rotated rx -179.9 ry 0 rz -90 deg; joints [13.502, -91.01, 136.581, -161.132, 46.195, 167.127]
  MoveL 3507 to (-311, 2.53, 6.83) mm, rotated rx -179.9 ry 0 rz -90 deg; joints [13.577, -90.887, 136.469, -161.034, 46.222, 167.063]
  MoveL 3508 to (-309.91, 2.45, 4.94) mm, rotated rx -179.9 ry 0 rz -90 deg; joints [13.612, -90.739, 136.333, -160.991, 46.241, 167.036]
  MoveL 3509 to (-309.55, 2.38, 2.79) mm, rotated rx -179.9 ry 0 rz -90 deg; joints [13.603, -90.586, 136.191, -161.007, 46.25, 167.05]
  MoveL 3510 to (-309.99, 2.3, 0.65) mm, rotated rx -179.9 ry 0 rz -90 deg; joints [13.55, -90.447, 136.063, -161.081, 46.248, 167.103]
  MoveL 3511 to (-311.16, 2.22, -1.19) mm, rotated rx -179.9 ry 0 rz -90 deg; joints [13.462, -90.339, 135.965, -161.202, 46.238, 167.188]
  MoveL 3512 to (-312.9, 2.15, -2.5) mm, rotated rx -179.9 ry 0 rz -90 deg; joints [13.35, -90.275, 135.911, -161.357, 46.222, 167.295]
  MoveL 3513 to (-315, 2.07, -3.1) mm, rotated rx -179.9 ry 0 rz -90 deg; joints [13.228, -90.264, 135.908, -161.524, 46.202, 167.41]
  MoveL 3514 to (-317.18, 1.99, -2.92) mm, rotated rx -179.9 ry 0 rz -90 deg; joints [13.112, -90.306, 135.956, -161.683, 46.183, 167.52]
  MoveL 3515 to (-319.14, 1.92, -1.97) mm, rotated rx -179.9 ry 0 rz -90 deg; joints [13.017, -90.396, 136.051, -161.813, 46.167, 167.61]
  MoveL 3516 to (-320.64, 1.84, -0.39) mm, rotated rx -179.9 ry 0 rz -90 deg; joints [12.955, -90.521, 136.18, -161.898, 46.157, 167.668]
  MoveL 3517 to (-321.48, 1.76, 1.63) mm, rotated rx -179.9 ry 0 rz -90 deg; joints [12.934, -90.665, 136.326, -161.926, 46.154, 167.688]
  MoveL 3518 to (-321.55, 1.69, 3.81) mm, rotated rx -179.9 ry 0 rz -90 deg; joints [12.958, -90.808, 136.47, -161.894, 46.161, 167.666]
  MoveL 3519 to (-320.84, 1.61, 5.87) mm, rotated rx -179.9 ry 0 rz -90 deg; joints [13.024, -90.932, 136.595, -161.806, 46.176, 167.606]
  MoveL 3520 to (-319.44, 1.53, 7.55) mm, rotated rx -179.9 ry 0 rz -90 deg; joints [13.123, -91.02, 136.685, -161.673, 46.199, 167.516]
  MoveL 3521 to (-317.53, 1.46, 8.61) mm, rotated rx -179.9 ry 0 rz -90 deg; joints [13.242, -91.058, 136.727, -161.513, 46.229, 167.409]
  MoveL 3522 to (-315.37, 1.38, 8.93) mm, rotated rx -179.9 ry 0 rz -90 deg; joints [13.365, -91.042, 136.716, -161.349, 46.262, 167.298]
  MoveL 3523 to (-313.24, 1.3, 8.46) mm, rotated rx -179.9 ry 0 rz -90 deg; joints [13.476, -90.973, 136.656, -161.201, 46.294, 167.2]
  MoveL 3524 to (-311.42, 1.23, 7.26) mm, rotated rx -179.9 ry 0 rz -90 deg; joints [13.561, -90.86, 136.552, -161.091, 46.323, 167.127]
  MoveL 3525 to (-310.14, 1.15, 5.49) mm, rotated rx -179.9 ry 0 rz -90 deg; joints [13.607, -90.718, 136.421, -161.031, 46.344, 167.09]
  MoveL 3526 to (-309.57, 1.07, 3.39) mm, rotated rx -179.9 ry 0 rz -90 deg; joints [13.61, -90.564, 136.279, -161.031, 46.355, 167.092]
  MoveL 3527 to (-309.79, 1, 1.22) mm, rotated rx -179.9 ry 0 rz -90 deg; joints [13.569, -90.42, 136.145, -161.089, 46.356, 167.135]
  MoveL 3528 to (-310.77, 0.92, -0.73) mm, rotated rx -179.9 ry 0 rz -90 deg; joints [13.49, -90.301, 136.037, -161.199, 46.348, 167.211]
  MoveL 3529 to (-312.38, 0.84, -2.21) mm, rotated rx -179.9 ry 0 rz -90 deg; joints [13.383, -90.225, 135.97, -161.346, 46.333, 167.313]
  MoveL 3530 to (-314.41, 0.77, -3.01) mm, rotated rx -179.9 ry 0 rz -90 deg; joints [13.262, -90.199, 135.953, -161.512, 46.314, 167.428]
  MoveL 3531 to (-316.59, 0.69, -3.05) mm, rotated rx -179.9 ry 0 rz -90 deg; joints [13.143, -90.227, 135.988, -161.675, 46.295, 167.54]
  MoveL 3532 to (-318.64, 0.61, -2.3) mm, rotated rx -179.9 ry 0 rz -90 deg; joints [13.04, -90.304, 136.071, -161.815, 46.278, 167.636]
  MoveL 3533 to (-320.29, 0.54, -0.87) mm, rotated rx -179.9 ry 0 rz -90 deg; joints [12.968, -90.421, 136.192, -161.913, 46.266, 167.704]
  MoveL 3534 to (-321.33, 0.46, 1.05) mm, rotated rx -179.9 ry 0 rz -90 deg; joints [12.936, -90.561, 136.335, -161.957, 46.262, 167.735]
  MoveL 3535 to (-321.61, 0.38, 3.21) mm, rotated rx -179.9 ry 0 rz -90 deg; joints [12.948, -90.707, 136.482, -161.942, 46.266, 167.725]
  MoveL 3536 to (-321.1, 0.31, 5.34) mm, rotated rx -179.9 ry 0 rz -90 deg; joints [13.003, -90.838, 136.614, -161.868, 46.279, 167.675]
  MoveL 3537 to (-319.88, 0.23, 7.14) mm, rotated rx -179.9 ry 0 rz -90 deg; joints [13.094, -90.937, 136.715, -161.746, 46.3, 167.592]
  MoveL 3538 to (-318.09, 0.15, 8.39) mm, rotated rx -179.9 ry 0 rz -90 deg; joints [13.209, -90.989, 136.77, -161.592, 46.328, 167.488]
  MoveL 3539 to (-315.97, 0.08, 8.92) mm, rotated rx -179.9 ry 0 rz -90 deg; joints [13.332, -90.988, 136.774, -161.427, 46.36, 167.377]
  MoveL 3540 to (-313.8, 0, 8.67) mm, rotated rx -179.9 ry 0 rz -90 deg; joints [13.448, -90.933, 136.727, -161.273, 46.393, 167.275]
  MoveL 3541 to (-313.76, 0, 8.65) mm, rotated rx -179.9 ry 0 rz -90 deg; joints [13.451, -90.932, 136.725, -161.27, 46.394, 167.273]
  MoveL 3542 to (-313.11, 0, 8.45) mm, rotated rx -179.9 ry 0 rz -90 deg; joints [13.484, -90.908, 136.702, -161.225, 46.402, 167.243]
  MoveC 3543 to (-309.55, 0, 5.45) mm, rotated rx -179.9 ry 0 rz -90 deg; joints [13.639, -90.65, 136.452, -161.018, 46.444, 167.105] to (-309.15, 0, 0.81) mm, rotated rx -179.9 ry 0 rz -90 deg; joints [13.599, -90.335, 136.146, -161.075, 46.444, 167.145]
  MoveL 3544 to (-309.15, 0, 0.81) mm, rotated rx -179.9 ry 0 rz -90 deg; joints [13.599, -90.335, 136.146, -161.075, 46.444, 167.145]
  MoveL 3545 to (-309.24, 0, 0.47) mm, rotated rx -179.9 ry 0 rz -90 deg; joints [13.59, -90.314, 136.125, -161.088, 46.442, 167.154]
  MoveL 3546 to (-309.31, 0, 0.13) mm, rotated rx -179.9 ry 0 rz -90 deg; joints [13.581, -90.292, 136.104, -161.1, 46.441, 167.162]
  MoveL 3547 to (-309.38, 0, -0.32) mm, rotated rx -179.9 ry 0 rz -90 deg; joints [13.572, -90.263, 136.076, -161.113, 46.44, 167.171]
  MoveL 3548 to (-309.41, 0, -0.77) mm, rotated rx -179.9 ry 0 rz -90 deg; joints [13.564, -90.234, 136.048, -161.123, 46.439, 167.179]
  MoveL 3549 to (-309.41, 0, -1.67) mm, rotated rx -179.9 ry 0 rz -90 deg; joints [13.552, -90.174, 135.99, -161.14, 46.438, 167.19]
  MoveL 3550 to (-309.41, 0, -310.57) mm, rotated rx -179.9 ry 0 rz -90 deg; joints [10.4, -71.298, 113.8, -164.541, 42.605, 168.878]
  MoveL 3551 to (-309.41, 0, -311.47) mm, rotated rx -179.9 ry 0 rz -90 deg; joints [10.393, -71.246, 113.729, -164.546, 42.585, 168.878]
  MoveL 3552 to (-309.38, 0, -311.92) mm, rotated rx -179.9 ry 0 rz -90 deg; joints [10.391, -71.219, 113.693, -164.546, 42.576, 168.876]
  MoveL 3553 to (-309.31, 0, -312.37) mm, rotated rx -179.9 ry 0 rz -90 deg; joints [10.39, -71.192, 113.656, -164.544, 42.566, 168.873]
  MoveL 3554 to (-309.24, 0, -312.7) mm, rotated rx -179.9 ry 0 rz -90 deg; joints [10.391, -71.172, 113.628, -164.541, 42.559, 168.87]
  MoveL 3555 to (-309.15, 0, -313.04) mm, rotated rx -179.9 ry 0 rz -90 deg; joints [10.392, -71.151, 113.6, -164.538, 42.552, 168.866]
  MoveL 3556 to (-309.08, 0, -313.26) mm, rotated rx -179.9 ry 0 rz -90 deg; joints [10.393, -71.138, 113.581, -164.534, 42.547, 168.862]
  MoveL 3557 to (-308.91, 0, -313.71) mm, rotated rx -179.9 ry 0 rz -90 deg; joints [10.397, -71.11, 113.543, -164.526, 42.538, 168.854]
  MoveL 3558 to (-308.7, 0, -314.16) mm, rotated rx -179.9 ry 0 rz -90 deg; joints [10.402, -71.081, 113.504, -164.515, 42.529, 168.844]
  MoveL 3559 to (-308.49, 0, -314.53) mm, rotated rx -179.9 ry 0 rz -90 deg; joints [10.408, -71.058, 113.472, -164.504, 42.521, 168.835]
  MoveL 3560 to (-308.25, 0, -314.9) mm, rotated rx -179.9 ry 0 rz -90 deg; joints [10.415, -71.034, 113.439, -164.491, 42.514, 168.823]
  MoveL 3561 to (-308.13, 0, -315.06) mm, rotated rx -179.9 ry 0 rz -90 deg; joints [10.419, -71.023, 113.424, -164.484, 42.511, 168.818]
  MoveL 3562 to (-307.96, 0, -315.27) mm, rotated rx -179.9 ry 0 rz -90 deg; joints [10.425, -71.009, 113.404, -164.474, 42.507, 168.81]
  MoveL 3563 to (-307.78, 0, -315.49) mm, rotated rx -179.9 ry 0 rz -90 deg; joints [10.431, -70.995, 113.384, -164.464, 42.503, 168.801]
  MoveL 3564 to (-307.57, 0, -315.7) mm, rotated rx -179.9 ry 0 rz -90 deg; joints [10.438, -70.98, 113.364, -164.452, 42.499, 168.792]
  MoveL 3565 to (-307.35, 0, -315.92) mm, rotated rx -179.9 ry 0 rz -90 deg; joints [10.445, -70.965, 113.344, -164.439, 42.495, 168.782]
  MoveL 3566 to (-307.31, 0, -315.96) mm, rotated rx -179.9 ry 0 rz -90 deg; joints [10.447, -70.962, 113.34, -164.437, 42.494, 168.779]
  MoveL 3567 to (-306.88, 0, -316.31) mm, rotated rx -179.9 ry 0 rz -90 deg; joints [10.462, -70.937, 113.306, -164.412, 42.488, 168.76]
  MoveL 3568 to (-306.45, 0, -316.6) mm, rotated rx -179.9 ry 0 rz -90 deg; joints [10.478, -70.916, 113.276, -164.387, 42.483, 168.74]
  MoveL 3569 to (-306.02, 0, -316.86) mm, rotated rx -179.9 ry 0 rz -90 deg; joints [10.494, -70.897, 113.249, -164.361, 42.48, 168.719]
  MoveL 3570 to (-305.55, 0, -317.08) mm, rotated rx -179.9 ry 0 rz -90 deg; joints [10.512, -70.879, 113.224, -164.333, 42.477, 168.698]
  MoveL 3571 to (-305.1, 0, -317.25) mm, rotated rx -179.9 ry 0 rz -90 deg; joints [10.53, -70.864, 113.204, -164.305, 42.474, 168.677]
  MoveL 3572 to (-304.66, 0, -317.38) mm, rotated rx -179.9 ry 0 rz -90 deg; joints [10.548, -70.851, 113.186, -164.278, 42.473, 168.656]
  MoveL 3573 to (-304.21, 0, -317.48) mm, rotated rx -179.9 ry 0 rz -90 deg; joints [10.566, -70.841, 113.172, -164.25, 42.473, 168.635]
  MoveL 3574 to (-303.76, 0, -317.55) mm, rotated rx -179.9 ry 0 rz -90 deg; joints [10.584, -70.832, 113.16, -164.223, 42.473, 168.614]
  MoveL 3575 to (-303.31, 0, -317.58) mm, rotated rx -179.9 ry 0 rz -90 deg; joints [10.603, -70.825, 113.15, -164.195, 42.474, 168.594]
  MoveL 3576 to (-302.86, 0, -317.59) mm, rotated rx -179.9 ry 0 rz -90 deg; joints [10.622, -70.82, 113.143, -164.166, 42.476, 168.573]
  MoveL 3577 to (315.44, 0, -317.59) mm, rotated rx -179.9 ry 0 rz -90 deg; joints [33.38, -56.807, 91.774, -130.221, 46.088, 141.471]
  MoveL 3578 to (315.89, 0, -317.58) mm, rotated rx -179.9 ry 0 rz -90 deg; joints [33.394, -56.793, 91.75, -130.199, 46.09, 141.451]
  MoveL 3579 to (316.34, 0, -317.54) mm, rotated rx -179.9 ry 0 rz -90 deg; joints [33.409, -56.779, 91.728, -130.177, 46.094, 141.431]
  MoveL 3580 to (316.79, 0, -317.47) mm, rotated rx -179.9 ry 0 rz -90 deg; joints [33.424, -56.768, 91.709, -130.155, 46.099, 141.412]
  MoveL 3581 to (317.24, 0, -317.36) mm, rotated rx -179.9 ry 0 rz -90 deg; joints [33.44, -56.758, 91.693, -130.134, 46.104, 141.394]
  MoveL 3582 to (317.69, 0, -317.23) mm, rotated rx -179.9 ry 0 rz -90 deg; joints [33.456, -56.75, 91.68, -130.112, 46.111, 141.376]
  MoveL 3583 to (318.14, 0, -317.05) mm, rotated rx -179.9 ry 0 rz -90 deg; joints [33.473, -56.744, 91.669, -130.09, 46.119, 141.359]
  MoveL 3584 to (318.54, 0, -316.86) mm, rotated rx -179.9 ry 0 rz -90 deg; joints [33.489, -56.74, 91.663, -130.071, 46.128, 141.345]
  MoveL 3585 to (318.78, 0, -316.72) mm, rotated rx -179.9 ry 0 rz -90 deg; joints [33.5, -56.739, 91.661, -130.059, 46.134, 141.336]
  MoveL 3586 to (319.03, 0, -316.56) mm, rotated rx -179.9 ry 0 rz -90 deg; joints [33.51, -56.738, 91.66, -130.047, 46.14, 141.328]
  MoveL 3587 to (319.43, 0, -316.28) mm, rotated rx -179.9 ry 0 rz -90 deg; joints [33.528, -56.739, 91.661, -130.028, 46.151, 141.315]
  MoveL 3588 to (319.83, 0, -315.96) mm, rotated rx -179.9 ry 0 rz -90 deg; joints [33.547, -56.743, 91.666, -130.009, 46.164, 141.303]
  MoveL 3589 to (319.93, 0, -315.86) mm, rotated rx -179.9 ry 0 rz -90 deg; joints [33.552, -56.744, 91.668, -130.004, 46.168, 141.3]
  MoveL 3590 to (320.14, 0, -315.66) mm, rotated rx -179.9 ry 0 rz -90 deg; joints [33.562, -56.748, 91.673, -129.995, 46.175, 141.295]
  MoveL 3591 to (320.32, 0, -315.46) mm, rotated rx -179.9 ry 0 rz -90 deg; joints [33.572, -56.752, 91.68, -129.986, 46.183, 141.29]
  MoveL 3592 to (320.65, 0, -315.06) mm, rotated rx -179.9 ry 0 rz -90 deg; joints [33.59, -56.761, 91.694, -129.97, 46.198, 141.282]
  MoveL 3593 to (320.83, 0, -314.8) mm, rotated rx -179.9 ry 0 rz -90 deg; joints [33.6, -56.768, 91.705, -129.962, 46.207, 141.279]
  MoveL 3594 to (321.04, 0, -314.48) mm, rotated rx -179.9 ry 0 rz -90 deg; joints [33.613, -56.778, 91.721, -129.952, 46.218, 141.275]
  MoveL 3595 to (321.22, 0, -314.16) mm, rotated rx -179.9 ry 0 rz -90 deg; joints [33.625, -56.788, 91.737, -129.944, 46.23, 141.273]
  MoveL 3596 to (321.43, 0, -313.71) mm, rotated rx -179.9 ry 0 rz -90 deg; joints [33.641, -56.804, 91.763, -129.934, 46.245, 141.272]
  MoveL 3597 to (321.6, 0, -313.26) mm, rotated rx -179.9 ry 0 rz -90 deg; joints [33.655, -56.822, 91.79, -129.926, 46.261, 141.272]
  MoveL 3598 to (321.73, 0, -312.81) mm, rotated rx -179.9 ry 0 rz -90 deg; joints [33.668, -56.841, 91.82, -129.92, 46.276, 141.274]
  MoveL 3599 to (321.83, 0, -312.37) mm, rotated rx -179.9 ry 0 rz -90 deg; joints [33.68, -56.861, 91.851, -129.915, 46.291, 141.278]
  MoveL 3600 to (321.89, 0, -311.92) mm, rotated rx -179.9 ry 0 rz -90 deg; joints [33.691, -56.882, 91.885, -129.912, 46.306, 141.283]
  MoveL 3601 to (321.93, 0, -311.47) mm, rotated rx -179.9 ry 0 rz -90 deg; joints [33.701, -56.904, 91.92, -129.911, 46.321, 141.289]
  MoveL 3602 to (321.93, 0, -310.57) mm, rotated rx -179.9 ry 0 rz -90 deg; joints [33.72, -56.95, 91.994, -129.911, 46.35, 141.305]
  MoveL 3603 to (321.93, 0, -1.67) mm, rotated rx -179.9 ry 0 rz -90 deg; joints [41.185, -71.705, 113.765, -126.774, 55.278, 143.716]
  MoveL 3604 to (321.93, 0, -0.77) mm, rotated rx -179.9 ry 0 rz -90 deg; joints [41.211, -71.745, 113.82, -126.757, 55.302, 143.716]
  MoveL 3605 to (321.89, 0, -0.32) mm, rotated rx -179.9 ry 0 rz -90 deg; joints [41.223, -71.767, 113.849, -126.749, 55.313, 143.717]
  MoveL 3606 to (321.83, 0, 0.13) mm, rotated rx -179.9 ry 0 rz -90 deg; joints [41.233, -71.789, 113.879, -126.743, 55.324, 143.719]
  MoveL 3607 to (321.73, 0, 0.58) mm, rotated rx -179.9 ry 0 rz -90 deg; joints [41.243, -71.813, 113.911, -126.739, 55.335, 143.722]
  MoveL 3608 to (321.6, 0, 1.03) mm, rotated rx -179.9 ry 0 rz -90 deg; joints [41.252, -71.839, 113.946, -126.735, 55.345, 143.726]
  MoveL 3609 to (321.43, 0, 1.48) mm, rotated rx -179.9 ry 0 rz -90 deg; joints [41.259, -71.865, 113.982, -126.733, 55.355, 143.731]
  MoveL 3610 to (321.22, 0, 1.93) mm, rotated rx -179.9 ry 0 rz -90 deg; joints [41.265, -71.894, 114.02, -126.733, 55.365, 143.738]
  MoveL 3611 to (321.04, 0, 2.25) mm, rotated rx -179.9 ry 0 rz -90 deg; joints [41.268, -71.915, 114.049, -126.734, 55.372, 143.743]
  MoveL 3612 to (320.83, 0, 2.57) mm, rotated rx -179.9 ry 0 rz -90 deg; joints [41.271, -71.937, 114.079, -126.736, 55.378, 143.75]
  MoveL 3613 to (320.65, 0, 2.82) mm, rotated rx -179.9 ry 0 rz -90 deg; joints [41.272, -71.956, 114.105, -126.738, 55.383, 143.755]
  MoveL 3614 to (320.32, 0, 3.22) mm, rotated rx -179.9 ry 0 rz -90 deg; joints [41.273, -71.986, 114.146, -126.743, 55.39, 143.766]
  MoveL 3615 to (320.14, 0, 3.42) mm, rotated rx -179.9 ry 0 rz -90 deg; joints [41.273, -72.002, 114.168, -126.747, 55.393, 143.771]
  MoveL 3616 to (319.93, 0, 3.62) mm, rotated rx -179.9 ry 0 rz -90 deg; joints [41.272, -72.019, 114.191, -126.751, 55.396, 143.778]
  MoveL 3617 to (319.83, 0, 3.72) mm, rotated rx -179.9 ry 0 rz -90 deg; joints [41.271, -72.028, 114.203, -126.754, 55.398, 143.781]
  MoveL 3618 to (319.43, 0, 4.05) mm, rotated rx -179.9 ry 0 rz -90 deg; joints [41.268, -72.058, 114.244, -126.763, 55.402, 143.794]
  MoveL 3619 to (319.03, 0, 4.33) mm, rotated rx -179.9 ry 0 rz -90 deg; joints [41.263, -72.086, 114.281, -126.773, 55.405, 143.806]
  MoveL 3620 to (318.79, 0, 4.48) mm, rotated rx -179.9 ry 0 rz -90 deg; joints [41.259, -72.102, 114.304, -126.78, 55.406, 143.814]
  MoveL 3621 to (318.54, 0, 4.62) mm, rotated rx -179.9 ry 0 rz -90 deg; joints [41.255, -72.118, 114.326, -126.787, 55.407, 143.822]
  MoveL 3622 to (318.14, 0, 4.81) mm, rotated rx -179.9 ry 0 rz -90 deg; joints [41.247, -72.142, 114.359, -126.8, 55.408, 143.834]
  MoveL 3623 to (317.69, 0, 4.99) mm, rotated rx -179.9 ry 0 rz -90 deg; joints [41.238, -72.168, 114.393, -126.814, 55.408, 143.849]
  MoveL 3624 to (317.24, 0, 5.13) mm, rotated rx -179.9 ry 0 rz -90 deg; joints [41.227, -72.191, 114.426, -126.829, 55.407, 143.863]
  MoveL 3625 to (316.79, 0, 5.23) mm, rotated rx -179.9 ry 0 rz -90 deg; joints [41.215, -72.213, 114.456, -126.845, 55.405, 143.877]
  MoveL 3626 to (316.34, 0, 5.3) mm, rotated rx -179.9 ry 0 rz -90 deg; joints [41.203, -72.234, 114.484, -126.862, 55.402, 143.891]
  MoveL 3627 to (315.89, 0, 5.34) mm, rotated rx -179.9 ry 0 rz -90 deg; joints [41.189, -72.253, 114.51, -126.879, 55.398, 143.906]
  MoveL 3628 to (315.44, 0, 5.35) mm, rotated rx -179.9 ry 0 rz -90 deg; joints [41.175, -72.271, 114.534, -126.897, 55.394, 143.92]
  MoveL 3629 to (-302.86, 0, 5.35) mm, rotated rx -179.9 ry 0 rz -90 deg; joints [14.004, -90.536, 136.337, -160.529, 46.527, 166.773]
  MoveL 3630 to (-303.31, 0, 5.35) mm, rotated rx -179.9 ry 0 rz -90 deg; joints [13.979, -90.543, 136.344, -160.562, 46.522, 166.796]
  MoveL 3631 to (-303.76, 0, 5.31) mm, rotated rx -179.9 ry 0 rz -90 deg; joints [13.954, -90.548, 136.349, -160.596, 46.516, 166.818]
  MoveL 3632 to (-304.21, 0, 5.25) mm, rotated rx -179.9 ry 0 rz -90 deg; joints [13.929, -90.551, 136.352, -160.63, 46.51, 166.842]
  MoveL 3633 to (-304.66, 0, 5.15) mm, rotated rx -179.9 ry 0 rz -90 deg; joints [13.903, -90.552, 136.353, -160.665, 46.504, 166.865]
  MoveL 3634 to (-305.1, 0, 5.01) mm, rotated rx -179.9 ry 0 rz -90 deg; joints [13.877, -90.55, 136.352, -160.7, 46.499, 166.889]
  MoveL 3635 to (-305.55, 0, 4.84) mm, rotated rx -179.9 ry 0 rz -90 deg; joints [13.85, -90.546, 136.348, -160.736, 46.493, 166.914]
  MoveL 3636 to (-306.02, 0, 4.62) mm, rotated rx -179.9 ry 0 rz -90 deg; joints [13.821, -90.538, 136.341, -160.774, 46.487, 166.94]
  MoveL 3637 to (-306.45, 0, 4.37) mm, rotated rx -179.9 ry 0 rz -90 deg; joints [13.794, -90.529, 136.332, -160.811, 46.481, 166.965]
  MoveL 3638 to (-306.88, 0, 4.07) mm, rotated rx -179.9 ry 0 rz -90 deg; joints [13.767, -90.516, 136.32, -160.848, 46.476, 166.99]
  MoveL 3639 to (-307.31, 0, 3.72) mm, rotated rx -179.9 ry 0 rz -90 deg; joints [13.739, -90.499, 136.304, -160.886, 46.47, 167.016]
  MoveL 3640 to (-307.35, 0, 3.68) mm, rotated rx -179.9 ry 0 rz -90 deg; joints [13.736, -90.497, 136.303, -160.89, 46.469, 167.019]
  MoveL 3641 to (-307.57, 0, 3.47) mm, rotated rx -179.9 ry 0 rz -90 deg; joints [13.721, -90.487, 136.292, -160.91, 46.466, 167.032]
  MoveL 3642 to (-307.78, 0, 3.25) mm, rotated rx -179.9 ry 0 rz -90 deg; joints [13.707, -90.476, 136.282, -160.929, 46.464, 167.045]
  MoveL 3643 to (-307.96, 0, 3.04) mm, rotated rx -179.9 ry 0 rz -90 deg; joints [13.694, -90.464, 136.271, -160.947, 46.461, 167.057]
  MoveL 3644 to (-308.13, 0, 2.82) mm, rotated rx -179.9 ry 0 rz -90 deg; joints [13.682, -90.453, 136.26, -160.963, 46.459, 167.069]
  MoveL 3645 to (-308.25, 0, 2.66) mm, rotated rx -179.9 ry 0 rz -90 deg; joints [13.673, -90.444, 136.251, -160.975, 46.457, 167.077]
  MoveL 3646 to (-308.49, 0, 2.29) mm, rotated rx -179.9 ry 0 rz -90 deg; joints [13.655, -90.423, 136.231, -160.999, 46.454, 167.093]
  MoveL 3647 to (-308.7, 0, 1.93) mm, rotated rx -179.9 ry 0 rz -90 deg; joints [13.639, -90.402, 136.211, -161.021, 46.451, 167.108]
  MoveL 3648 to (-308.91, 0, 1.48) mm, rotated rx -179.9 ry 0 rz -90 deg; joints [13.621, -90.375, 136.185, -161.045, 46.448, 167.125]
  MoveL 3649 to (-309.08, 0, 1.03) mm, rotated rx -179.9 ry 0 rz -90 deg; joints [13.606, -90.348, 136.159, -161.066, 46.445, 167.139]
  MoveL 3650 to (-309.15, 0, 0.81) mm, rotated rx -179.9 ry 0 rz -90 deg; joints [13.599, -90.335, 136.146, -161.075, 46.444, 167.145]
  MoveC 3651 to (-309.77, 0, 0.07) mm, rotated rx -179.9 ry 0 rz -90 deg; joints [13.555, -90.295, 136.108, -161.135, 46.435, 167.186] to (-310.74, 0, -0.02) mm, rotated rx -179.9 ry 0 rz -90 deg; joints [13.501, -90.305, 136.118, -161.207, 46.424, 167.235]
  MoveL 3652 to (-310.74, 0, -0.02) mm, rotated rx -179.9 ry 0 rz -90 deg; joints [13.501, -90.305, 136.118, -161.207, 46.424, 167.235]
  MoveC 3653 to (-310.77, 0, -0.01) mm, rotated rx -179.9 ry 0 rz -90 deg; joints [13.5, -90.306, 136.119, -161.209, 46.423, 167.237] to (-310.8, 0, 0) mm, rotated rx -179.9 ry 0 rz -90 deg; joints [13.498, -90.307, 136.12, -161.211, 46.423, 167.238]
  MoveL 3654 to (-310.8, 0, 0) mm, rotated rx -179.9 ry 0 rz -90 deg; joints [13.498, -90.307, 136.12, -161.211, 46.423, 167.238]
  MoveL 3655 to (-325.34, 0, 3.85) mm, rotated rx -179.9 ry 0 rz -90 deg; joints [12.751, -90.788, 136.594, -162.218, 46.253, 167.919]
  MoveC 3656 to (-327.44, 0, 4.87) mm, rotated rx -179.9 ry 0 rz -90 deg; joints [12.648, -90.888, 136.691, -162.356, 46.229, 168.013] to (-328.99, 0, 6.62) mm, rotated rx -179.9 ry 0 rz -90 deg; joints [12.584, -91.028, 136.827, -162.441, 46.211, 168.07]
  MoveL 3657 to (-328.99, 0, 6.62) mm, rotated rx -179.9 ry 0 rz -90 deg; joints [12.584, -91.028, 136.827, -162.441, 46.211, 168.07]
  MoveL 3658 to (-329.02, 0, 6.66) mm, rotated rx -179.9 ry 0 rz -90 deg; joints [12.583, -91.031, 136.83, -162.442, 46.211, 168.07]
  MoveL 3659 to (-329.75, -0.08, 8.69) mm, rotated rx -179.9 ry 0 rz -90 deg; joints [12.568, -91.176, 136.975, -162.463, 46.208, 168.084]
  MoveL 3660 to (-329.71, -0.15, 10.86) mm, rotated rx -179.9 ry 0 rz -90 deg; joints [12.597, -91.318, 137.117, -162.424, 46.213, 168.058]
  MoveL 3661 to (-328.92, -0.23, 12.87) mm, rotated rx -179.9 ry 0 rz -90 deg; joints [12.666, -91.438, 137.237, -162.33, 46.228, 167.994]
  MoveL 3662 to (-327.47, -0.3, 14.47) mm, rotated rx -179.9 ry 0 rz -90 deg; joints [12.768, -91.522, 137.321, -162.193, 46.25, 167.901]
  MoveL 3663 to (-325.54, -0.38, 15.46) mm, rotated rx -179.9 ry 0 rz -90 deg; joints [12.887, -91.556, 137.358, -162.032, 46.279, 167.792]
  MoveL 3664 to (-323.39, -0.46, 15.7) mm, rotated rx -179.9 ry 0 rz -90 deg; joints [13.01, -91.535, 137.344, -161.868, 46.312, 167.682]
  MoveL 3665 to (-321.29, -0.53, 15.17) mm, rotated rx -179.9 ry 0 rz -90 deg; joints [13.12, -91.463, 137.281, -161.723, 46.344, 167.586]
  MoveL 3666 to (-319.52, -0.61, 13.94) mm, rotated rx -179.9 ry 0 rz -90 deg; joints [13.202, -91.348, 137.178, -161.615, 46.373, 167.515]
  MoveL 3667 to (-318.29, -0.68, 12.15) mm, rotated rx -179.9 ry 0 rz -90 deg; joints [13.247, -91.205, 137.047, -161.558, 46.394, 167.48]
  MoveL 3668 to (-317.78, -0.76, 10.05) mm, rotated rx -179.9 ry 0 rz -90 deg; joints [13.248, -91.052, 136.907, -161.561, 46.407, 167.485]
  MoveL 3669 to (-318.03, -0.84, 7.9) mm, rotated rx -179.9 ry 0 rz -90 deg; joints [13.206, -90.908, 136.775, -161.622, 46.409, 167.529]
  MoveL 3670 to (-319.03, -0.91, 5.98) mm, rotated rx -179.9 ry 0 rz -90 deg; joints [13.126, -90.791, 136.67, -161.733, 46.403, 167.606]
  MoveL 3671 to (-320.64, -0.99, 4.54) mm, rotated rx -179.9 ry 0 rz -90 deg; joints [13.019, -90.715, 136.604, -161.88, 46.389, 167.709]
  MoveL 3672 to (-322.66, -1.06, 3.76) mm, rotated rx -179.9 ry 0 rz -90 deg; joints [12.898, -90.69, 136.587, -162.046, 46.371, 167.823]
  MoveL 3673 to (-324.82, -1.14, 3.74) mm, rotated rx -179.9 ry 0 rz -90 deg; joints [12.779, -90.717, 136.622, -162.209, 46.352, 167.935]
  MoveL 3674 to (-326.85, -1.22, 4.48) mm, rotated rx -179.9 ry 0 rz -90 deg; joints [12.676, -90.794, 136.703, -162.349, 46.335, 168.031]
  MoveL 3675 to (-328.49, -1.29, 5.9) mm, rotated rx -179.9 ry 0 rz -90 deg; joints [12.603, -90.91, 136.822, -162.448, 46.323, 168.099]
  MoveL 3676 to (-329.53, -1.37, 7.8) mm, rotated rx -179.9 ry 0 rz -90 deg; joints [12.57, -91.049, 136.962, -162.494, 46.317, 168.13]
  MoveL 3677 to (-329.82, -1.44, 9.94) mm, rotated rx -179.9 ry 0 rz -90 deg; joints [12.58, -91.195, 137.108, -162.48, 46.319, 168.121]
  MoveL 3678 to (-329.35, -1.52, 12.05) mm, rotated rx -179.9 ry 0 rz -90 deg; joints [12.633, -91.327, 137.239, -162.408, 46.33, 168.072]
  MoveL 3679 to (-328.15, -1.6, 13.85) mm, rotated rx -179.9 ry 0 rz -90 deg; joints [12.722, -91.427, 137.341, -162.288, 46.349, 167.991]
  MoveL 3680 to (-326.4, -1.67, 15.12) mm, rotated rx -179.9 ry 0 rz -90 deg; joints [12.836, -91.483, 137.399, -162.135, 46.375, 167.888]
  MoveL 3681 to (-324.31, -1.75, 15.69) mm, rotated rx -179.9 ry 0 rz -90 deg; joints [12.959, -91.486, 137.407, -161.97, 46.407, 167.777]
  MoveL 3682 to (-322.16, -1.82, 15.49) mm, rotated rx -179.9 ry 0 rz -90 deg; joints [13.076, -91.436, 137.364, -161.814, 46.439, 167.673]
  MoveL 3683 to (-320.22, -1.9, 14.54) mm, rotated rx -179.9 ry 0 rz -90 deg; joints [13.172, -91.337, 137.276, -161.688, 46.47, 167.59]
  MoveL 3684 to (-318.73, -1.97, 12.96) mm, rotated rx -179.9 ry 0 rz -90 deg; joints [13.234, -91.204, 137.155, -161.609, 46.494, 167.539]
  MoveL 3685 to (-317.9, -2.05, 10.97) mm, rotated rx -179.9 ry 0 rz -90 deg; joints [13.254, -91.053, 137.016, -161.586, 46.511, 167.527]
  MoveL 3686 to (-317.83, -2.13, 8.8) mm, rotated rx -179.9 ry 0 rz -90 deg; joints [13.229, -90.903, 136.879, -161.622, 46.518, 167.554]
  MoveL 3687 to (-318.52, -2.2, 6.75) mm, rotated rx -179.9 ry 0 rz -90 deg; joints [13.165, -90.773, 136.76, -161.713, 46.515, 167.618]
  MoveL 3688 to (-319.89, -2.28, 5.08) mm, rotated rx -179.9 ry 0 rz -90 deg; joints [13.067, -90.678, 136.676, -161.847, 46.504, 167.711]
  MoveL 3689 to (-321.77, -2.35, 4) mm, rotated rx -179.9 ry 0 rz -90 deg; joints [12.95, -90.63, 136.638, -162.007, 46.487, 167.822]
  MoveL 3690 to (-323.9, -2.43, 3.65) mm, rotated rx -179.9 ry 0 rz -90 deg; joints [12.829, -90.635, 136.65, -162.174, 46.468, 167.936]
  MoveL 3691 to (-326.02, -2.51, 4.08) mm, rotated rx -179.9 ry 0 rz -90 deg; joints [12.717, -90.692, 136.713, -162.325, 46.45, 168.04]
  MoveL 3692 to (-327.86, -2.58, 5.22) mm, rotated rx -179.9 ry 0 rz -90 deg; joints [12.63, -90.793, 136.817, -162.444, 46.436, 168.121]
  MoveL 3693 to (-329.17, -2.66, 6.94) mm, rotated rx -179.9 ry 0 rz -90 deg; joints [12.579, -90.924, 136.951, -162.513, 46.427, 168.169]
  MoveL 3694 to (-329.79, -2.73, 9.02) mm, rotated rx -179.9 ry 0 rz -90 deg; joints [12.571, -91.069, 137.096, -162.525, 46.426, 168.177]
  MoveL 3695 to (-329.64, -2.81, 11.17) mm, rotated rx -179.9 ry 0 rz -90 deg; joints [12.606, -91.209, 137.236, -162.477, 46.433, 168.144]
  MoveL 3696 to (-328.74, -2.89, 13.14) mm, rotated rx -179.9 ry 0 rz -90 deg; joints [12.681, -91.325, 137.352, -162.376, 46.449, 168.076]
  MoveL 3697 to (-327.2, -2.96, 14.66) mm, rotated rx -179.9 ry 0 rz -90 deg; joints [12.786, -91.401, 137.43, -162.235, 46.473, 167.981]
  MoveL 3698 to (-325.23, -3.04, 15.54) mm, rotated rx -179.9 ry 0 rz -90 deg; joints [12.907, -91.427, 137.46, -162.073, 46.502, 167.872]
  MoveL 3699 to (-323.07, -3.11, 15.67) mm, rotated rx -179.9 ry 0 rz -90 deg; joints [13.029, -91.399, 137.438, -161.911, 46.534, 167.764]
  MoveL 3700 to (-321, -3.19, 15.03) mm, rotated rx -179.9 ry 0 rz -90 deg; joints [13.136, -91.32, 137.368, -161.77, 46.566, 167.671]
  MoveL 3701 to (-319.29, -3.27, 13.7) mm, rotated rx -179.9 ry 0 rz -90 deg; joints [13.213, -91.2, 137.259, -161.67, 46.593, 167.606]
  MoveL 3702 to (-318.17, -3.34, 11.85) mm, rotated rx -179.9 ry 0 rz -90 deg; joints [13.251, -91.054, 137.126, -161.622, 46.613, 167.576]
  MoveL 3703 to (-317.76, -3.42, 9.73) mm, rotated rx -179.9 ry 0 rz -90 deg; joints [13.246, -90.901, 136.985, -161.633, 46.624, 167.587]
  MoveL 3704 to (-318.14, -3.49, 7.59) mm, rotated rx -179.9 ry 0 rz -90 deg; joints [13.197, -90.76, 136.857, -161.702, 46.625, 167.636]
  MoveL 3705 to (-319.24, -3.57, 5.73) mm, rotated rx -179.9 ry 0 rz -90 deg; joints [13.112, -90.649, 136.756, -161.819, 46.617, 167.717]
  MoveL 3706 to (-320.93, -3.65, 4.38) mm, rotated rx -179.9 ry 0 rz -90 deg; joints [13.002, -90.58, 136.697, -161.97, 46.603, 167.821]
  MoveL 3707 to (-322.98, -3.72, 3.71) mm, rotated rx -179.9 ry 0 rz -90 deg; joints [12.881, -90.563, 136.688, -162.136, 46.585, 167.935]
  MoveL 3708 to (-325.14, -3.8, 3.8) mm, rotated rx -179.9 ry 0 rz -90 deg; joints [12.763, -90.598, 136.73, -162.296, 46.566, 168.045]
  MoveL 3709 to (-327.13, -3.87, 4.66) mm, rotated rx -179.9 ry 0 rz -90 deg; joints [12.664, -90.681, 136.818, -162.431, 46.55, 168.137]
  MoveL 3710 to (-328.69, -3.95, 6.15) mm, rotated rx -179.9 ry 0 rz -90 deg; joints [12.596, -90.801, 136.941, -162.522, 46.538, 168.2]
  MoveL 3711 to (-329.62, -4.03, 8.11) mm, rotated rx -179.9 ry 0 rz -90 deg; joints [12.569, -90.943, 137.084, -162.559, 46.534, 168.225]
  MoveL 3712 to (-329.8, -4.1, 10.26) mm, rotated rx -179.9 ry 0 rz -90 deg; joints [12.586, -91.087, 137.228, -162.536, 46.538, 168.21]
  MoveL 3713 to (-329.21, -4.18, 12.35) mm, rotated rx -179.9 ry 0 rz -90 deg; joints [12.645, -91.215, 137.357, -162.457, 46.55, 168.156]
  MoveL 3714 to (-327.92, -4.25, 14.08) mm, rotated rx -179.9 ry 0 rz -90 deg; joints [12.739, -91.31, 137.452, -162.331, 46.571, 168.071]
  MoveL 3715 to (-326.1, -4.33, 15.26) mm, rotated rx -179.9 ry 0 rz -90 deg; joints [12.855, -91.358, 137.503, -162.176, 46.598, 167.967]
  MoveL 3716 to (-323.99, -4.4, 15.71) mm, rotated rx -179.9 ry 0 rz -90 deg; joints [12.979, -91.353, 137.503, -162.011, 46.63, 167.857]
  MoveL 3717 to (-321.85, -4.48, 15.39) mm, rotated rx -179.9 ry 0 rz -90 deg; joints [13.094, -91.294, 137.453, -161.859, 46.662, 167.756]
  MoveL 3718 to (-319.96, -4.56, 14.34) mm, rotated rx -179.9 ry 0 rz -90 deg; joints [13.185, -91.19, 137.359, -161.74, 46.691, 167.678]
  MoveL 3719 to (-318.56, -4.63, 12.68) mm, rotated rx -179.9 ry 0 rz -90 deg; joints [13.241, -91.053, 137.234, -161.668, 46.714, 167.633]
  MoveL 3720 to (-317.84, -4.71, 10.65) mm, rotated rx -179.9 ry 0 rz -90 deg; joints [13.254, -90.901, 137.094, -161.654, 46.729, 167.626]
  MoveL 3721 to (-317.88, -4.78, 8.48) mm, rotated rx -179.9 ry 0 rz -90 deg; joints [13.223, -90.753, 136.958, -161.699, 46.734, 167.659]
  MoveL 3722 to (-318.69, -4.86, 6.47) mm, rotated rx -179.9 ry 0 rz -90 deg; joints [13.153, -90.627, 136.844, -161.797, 46.729, 167.728]
  MoveL 3723 to (-320.15, -4.94, 4.88) mm, rotated rx -179.9 ry 0 rz -90 deg; joints [13.052, -90.539, 136.766, -161.935, 46.718, 167.823]
  MoveL 3724 to (-322.08, -5.01, 3.9) mm, rotated rx -179.9 ry 0 rz -90 deg; joints [12.933, -90.499, 136.735, -162.097, 46.701, 167.934]
  MoveL 3725 to (-324.23, -5.09, 3.67) mm, rotated rx -179.9 ry 0 rz -90 deg; joints [12.812, -90.512, 136.755, -162.262, 46.682, 168.047]
  MoveL 3726 to (-326.32, -5.16, 4.21) mm, rotated rx -179.9 ry 0 rz -90 deg; joints [12.703, -90.576, 136.825, -162.409, 46.664, 168.148]
  MoveL 3727 to (-328.09, -5.24, 5.45) mm, rotated rx -179.9 ry 0 rz -90 deg; joints [12.621, -90.682, 136.935, -162.521, 46.651, 168.224]
  MoveL 3728 to (-329.31, -5.32, 7.24) mm, rotated rx -179.9 ry 0 rz -90 deg; joints [12.576, -90.817, 137.071, -162.582, 46.644, 168.266]
  MoveL 3729 to (-329.82, -5.39, 9.34) mm, rotated rx -179.9 ry 0 rz -90 deg; joints [12.574, -90.962, 137.217, -162.585, 46.644, 168.268]
  MoveL 3730 to (-329.55, -5.47, 11.49) mm, rotated rx -179.9 ry 0 rz -90 deg; joints [12.616, -91.099, 137.355, -162.529, 46.653, 168.23]
  MoveL 3731 to (-328.55, -5.54, 13.4) mm, rotated rx -179.9 ry 0 rz -90 deg; joints [12.696, -91.21, 137.466, -162.421, 46.67, 168.158]
  MoveL 3732 to (-326.93, -5.62, 14.84) mm, rotated rx -179.9 ry 0 rz -90 deg; joints [12.804, -91.279, 137.537, -162.276, 46.695, 168.06]
  MoveL 3733 to (-324.91, -5.7, 15.61) mm, rotated rx -179.9 ry 0 rz -90 deg; joints [12.927, -91.297, 137.559, -162.113, 46.725, 167.951]
  MoveL 3734 to (-322.74, -5.77, 15.62) mm, rotated rx -179.9 ry 0 rz -90 deg; joints [13.047, -91.26, 137.53, -161.953, 46.757, 167.845]
  MoveL 3735 to (-320.72, -5.85, 14.87) mm, rotated rx -179.9 ry 0 rz -90 deg; joints [13.15, -91.174, 137.453, -161.818, 46.788, 167.756]
  MoveL 3736 to (-319.08, -5.92, 13.45) mm, rotated rx -179.9 ry 0 rz -90 deg; joints [13.222, -91.05, 137.339, -161.725, 46.814, 167.696]
  MoveL 3737 to (-318.06, -6, 11.54) mm, rotated rx -179.9 ry 0 rz -90 deg; joints [13.254, -90.902, 137.204, -161.686, 46.832, 167.673]
  MoveL 3738 to (-318.04, -6, 11.5) mm, rotated rx -179.9 ry 0 rz -90 deg; joints [13.254, -90.899, 137.201, -161.686, 46.833, 167.673]
  MoveL 3739 to (-317.84, -6, 10.85) mm, rotated rx -179.9 ry 0 rz -90 deg; joints [13.257, -90.852, 137.155, -161.682, 46.835, 167.671]
  MoveC 3740 to (-318.24, -6, 6.21) mm, rotated rx -179.9 ry 0 rz -90 deg; joints [13.175, -90.547, 136.862, -161.796, 46.828, 167.75] to (-321.8, -6, 3.21) mm, rotated rx -179.9 ry 0 rz -90 deg; joints [12.94, -90.401, 136.723, -162.113, 46.784, 167.964]
  MoveL 3741 to (-321.8, -6, 3.21) mm, rotated rx -179.9 ry 0 rz -90 deg; joints [12.94, -90.401, 136.723, -162.113, 46.784, 167.964]
  MoveL 3742 to (-324.43, -6, 2.39) mm, rotated rx -179.9 ry 0 rz -90 deg; joints [12.785, -90.385, 136.709, -162.321, 46.753, 168.105]
  MoveL 3743 to (-325.33, -6, 2.09) mm, rotated rx -179.9 ry 0 rz -90 deg; joints [12.732, -90.379, 136.704, -162.392, 46.743, 168.153]
  MoveL 3744 to (-325.72, -6, 1.93) mm, rotated rx -179.9 ry 0 rz -90 deg; joints [12.709, -90.374, 136.699, -162.424, 46.738, 168.175]
  MoveL 3745 to (-325.97, -6, 1.8) mm, rotated rx -179.9 ry 0 rz -90 deg; joints [12.693, -90.369, 136.695, -162.445, 46.735, 168.189]
  MoveL 3746 to (-326.22, -6, 1.66) mm, rotated rx -179.9 ry 0 rz -90 deg; joints [12.677, -90.364, 136.689, -162.466, 46.733, 168.203]
  MoveL 3747 to (-326.45, -6, 1.53) mm, rotated rx -179.9 ry 0 rz -90 deg; joints [12.663, -90.358, 136.684, -162.485, 46.73, 168.216]
  MoveL 3748 to (-326.67, -6, 1.38) mm, rotated rx -179.9 ry 0 rz -90 deg; joints [12.649, -90.352, 136.678, -162.504, 46.727, 168.229]
  MoveL 3749 to (-326.9, -6, 1.22) mm, rotated rx -179.9 ry 0 rz -90 deg; joints [12.635, -90.344, 136.671, -162.524, 46.725, 168.242]
  MoveL 3750 to (-327.12, -6, 1.04) mm, rotated rx -179.9 ry 0 rz -90 deg; joints [12.62, -90.335, 136.662, -162.543, 46.722, 168.255]
  MoveL 3751 to (-327.14, -6, 1.03) mm, rotated rx -179.9 ry 0 rz -90 deg; joints [12.619, -90.335, 136.662, -162.545, 46.722, 168.256]
  MoveL 3752 to (-327.38, -6, 0.82) mm, rotated rx -179.9 ry 0 rz -90 deg; joints [12.603, -90.324, 136.652, -162.566, 46.719, 168.271]
  MoveL 3753 to (-327.62, -6, 0.58) mm, rotated rx -179.9 ry 0 rz -90 deg; joints [12.587, -90.312, 136.64, -162.588, 46.716, 168.286]
  MoveL 3754 to (-327.83, -6, 0.35) mm, rotated rx -179.9 ry 0 rz -90 deg; joints [12.573, -90.3, 136.628, -162.607, 46.714, 168.299]
  MoveL 3755 to (-328.02, -6, 0.13) mm, rotated rx -179.9 ry 0 rz -90 deg; joints [12.56, -90.288, 136.616, -162.625, 46.711, 168.311]
  MoveL 3756 to (-328.02, -6, 0.12) mm, rotated rx -179.9 ry 0 rz -90 deg; joints [12.559, -90.287, 136.616, -162.626, 46.711, 168.311]
  MoveL 3757 to (-328.19, -6, -0.1) mm, rotated rx -179.9 ry 0 rz -90 deg; joints [12.547, -90.275, 136.604, -162.642, 46.709, 168.322]
  MoveL 3758 to (-328.35, -6, -0.32) mm, rotated rx -179.9 ry 0 rz -90 deg; joints [12.536, -90.262, 136.592, -162.657, 46.707, 168.333]
  MoveL 3759 to (-328.62, -6, -0.77) mm, rotated rx -179.9 ry 0 rz -90 deg; joints [12.516, -90.237, 136.567, -162.685, 46.704, 168.352]
  MoveL 3760 to (-328.78, -6, -1.08) mm, rotated rx -179.9 ry 0 rz -90 deg; joints [12.503, -90.218, 136.549, -162.702, 46.702, 168.363]
  MoveL 3761 to (-328.92, -6, -1.39) mm, rotated rx -179.9 ry 0 rz -90 deg; joints [12.491, -90.199, 136.531, -162.718, 46.7, 168.374]
  MoveL 3762 to (-329.03, -6, -1.67) mm, rotated rx -179.9 ry 0 rz -90 deg; joints [12.482, -90.183, 136.515, -162.73, 46.699, 168.383]
  MoveL 3763 to (-329.17, -6, -2.11) mm, rotated rx -179.9 ry 0 rz -90 deg; joints [12.469, -90.155, 136.488, -162.749, 46.696, 168.395]
  MoveL 3764 to (-329.28, -6, -2.56) mm, rotated rx -179.9 ry 0 rz -90 deg; joints [12.457, -90.126, 136.46, -162.764, 46.695, 168.406]
  MoveL 3765 to (-329.36, -6, -3.01) mm, rotated rx -179.9 ry 0 rz -90 deg; joints [12.448, -90.097, 136.432, -162.778, 46.694, 168.415]
  MoveL 3766 to (-329.4, -6, -3.46) mm, rotated rx -179.9 ry 0 rz -90 deg; joints [12.44, -90.068, 136.403, -162.788, 46.693, 168.422]
  MoveL 3767 to (-329.41, -6, -4.36) mm, rotated rx -179.9 ry 0 rz -90 deg; joints [12.428, -90.008, 136.345, -162.804, 46.691, 168.433]
  MoveL 3768 to (-329.41, -6, -310.57) mm, rotated rx -179.9 ry 0 rz -90 deg; joints [9.549, -71.28, 114.272, -165.907, 42.919, 169.952]
  MoveL 3769 to (-329.41, -6, -311.47) mm, rotated rx -179.9 ry 0 rz -90 deg; joints [9.543, -71.227, 114.2, -165.911, 42.899, 169.952]
  MoveL 3770 to (-329.38, -6, -311.92) mm, rotated rx -179.9 ry 0 rz -90 deg; joints [9.541, -71.201, 114.164, -165.911, 42.89, 169.95]
  MoveL 3771 to (-329.31, -6, -312.37) mm, rotated rx -179.9 ry 0 rz -90 deg; joints [9.54, -71.174, 114.127, -165.91, 42.88, 169.947]
  MoveL 3772 to (-329.21, -6, -312.81) mm, rotated rx -179.9 ry 0 rz -90 deg; joints [9.541, -71.147, 114.09, -165.906, 42.87, 169.943]
  MoveL 3773 to (-329.08, -6, -313.26) mm, rotated rx -179.9 ry 0 rz -90 deg; joints [9.544, -71.12, 114.053, -165.899, 42.861, 169.936]
  MoveL 3774 to (-328.92, -6, -313.69) mm, rotated rx -179.9 ry 0 rz -90 deg; joints [9.547, -71.094, 114.017, -165.891, 42.852, 169.929]
  MoveL 3775 to (-328.7, -6, -314.16) mm, rotated rx -179.9 ry 0 rz -90 deg; joints [9.554, -71.064, 113.976, -165.88, 42.842, 169.919]
  MoveL 3776 to (-328.44, -6, -314.61) mm, rotated rx -179.9 ry 0 rz -90 deg; joints [9.561, -71.035, 113.937, -165.866, 42.833, 169.907]
  MoveL 3777 to (-328.13, -6, -315.06) mm, rotated rx -179.9 ry 0 rz -90 deg; joints [9.571, -71.006, 113.896, -165.849, 42.824, 169.892]
  MoveL 3778 to (-328.02, -6, -315.2) mm, rotated rx -179.9 ry 0 rz -90 deg; joints [9.575, -70.997, 113.884, -165.842, 42.822, 169.887]
  MoveL 3779 to (-327.69, -6, -315.58) mm, rotated rx -179.9 ry 0 rz -90 deg; joints [9.586, -70.972, 113.849, -165.824, 42.814, 169.872]
  MoveL 3780 to (-327.31, -6, -315.96) mm, rotated rx -179.9 ry 0 rz -90 deg; joints [9.6, -70.946, 113.813, -165.801, 42.807, 169.854]
  MoveL 3781 to (-327.12, -6, -316.12) mm, rotated rx -179.9 ry 0 rz -90 deg; joints [9.606, -70.935, 113.798, -165.79, 42.805, 169.846]
  MoveL 3782 to (-326.9, -6, -316.3) mm, rotated rx -179.9 ry 0 rz -90 deg; joints [9.615, -70.923, 113.781, -165.777, 42.801, 169.835]
  MoveL 3783 to (-326.67, -6, -316.46) mm, rotated rx -179.9 ry 0 rz -90 deg; joints [9.623, -70.911, 113.765, -165.764, 42.799, 169.825]
  MoveL 3784 to (-326.45, -6, -316.61) mm, rotated rx -179.9 ry 0 rz -90 deg; joints [9.632, -70.9, 113.75, -165.75, 42.796, 169.815]
  MoveL 3785 to (-326.22, -6, -316.74) mm, rotated rx -179.9 ry 0 rz -90 deg; joints [9.64, -70.89, 113.736, -165.737, 42.794, 169.804]
  MoveL 3786 to (-326.02, -6, -316.86) mm, rotated rx -179.9 ry 0 rz -90 deg; joints [9.648, -70.882, 113.724, -165.725, 42.792, 169.795]
  MoveL 3787 to (-325.67, -6, -317.02) mm, rotated rx -179.9 ry 0 rz -90 deg; joints [9.661, -70.868, 113.706, -165.704, 42.789, 169.779]
  MoveL 3788 to (-325.33, -6, -317.17) mm, rotated rx -179.9 ry 0 rz -90 deg; joints [9.675, -70.857, 113.689, -165.683, 42.788, 169.763]
  MoveL 3789 to (-324.88, -6, -317.32) mm, rotated rx -179.9 ry 0 rz -90 deg; joints [9.693, -70.843, 113.671, -165.655, 42.786, 169.742]
  MoveL 3790 to (-324.43, -6, -317.44) mm, rotated rx -179.9 ry 0 rz -90 deg; joints [9.711, -70.832, 113.655, -165.628, 42.785, 169.721]
  MoveL 3791 to (-323.98, -6, -317.52) mm, rotated rx -179.9 ry 0 rz -90 deg; joints [9.73, -70.823, 113.642, -165.6, 42.785, 169.701]
  MoveL 3792 to (-323.53, -6, -317.57) mm, rotated rx -179.9 ry 0 rz -90 deg; joints [9.749, -70.816, 113.632, -165.572, 42.785, 169.68]
  MoveL 3793 to (-322.63, -6, -317.59) mm, rotated rx -179.9 ry 0 rz -90 deg; joints [9.787, -70.806, 113.618, -165.516, 42.788, 169.639]
  MoveL 3794 to (324.43, -6, -317.59) mm, rotated rx -179.9 ry 0 rz -90 deg; joints [33.656, -56.333, 91.457, -130.039, 46.362, 141.437]
  MoveL 3795 to (325.33, -6, -317.58) mm, rotated rx -179.9 ry 0 rz -90 deg; joints [33.683, -56.302, 91.407, -129.996, 46.367, 141.397]
  MoveL 3796 to (325.77, -6, -317.55) mm, rotated rx -179.9 ry 0 rz -90 deg; joints [33.697, -56.288, 91.385, -129.974, 46.37, 141.377]
  MoveL 3797 to (326.22, -6, -317.49) mm, rotated rx -179.9 ry 0 rz -90 deg; joints [33.712, -56.276, 91.365, -129.953, 46.374, 141.358]
  MoveL 3798 to (326.67, -6, -317.39) mm, rotated rx -179.9 ry 0 rz -90 deg; joints [33.728, -56.266, 91.348, -129.931, 46.38, 141.34]
  MoveL 3799 to (327.12, -6, -317.26) mm, rotated rx -179.9 ry 0 rz -90 deg; joints [33.744, -56.257, 91.334, -129.909, 46.386, 141.322]
  MoveL 3800 to (327.57, -6, -317.09) mm, rotated rx -179.9 ry 0 rz -90 deg; joints [33.761, -56.251, 91.323, -129.888, 46.394, 141.305]
  MoveL 3801 to (328.02, -6, -316.88) mm, rotated rx -179.9 ry 0 rz -90 deg; joints [33.779, -56.246, 91.315, -129.866, 46.403, 141.289]
  MoveL 3802 to (328.06, -6, -316.86) mm, rotated rx -179.9 ry 0 rz -90 deg; joints [33.78, -56.246, 91.314, -129.864, 46.404, 141.287]
  MoveL 3803 to (328.49, -6, -316.61) mm, rotated rx -179.9 ry 0 rz -90 deg; joints [33.798, -56.244, 91.311, -129.844, 46.414, 141.273]
  MoveL 3804 to (328.92, -6, -316.31) mm, rotated rx -179.9 ry 0 rz -90 deg; joints [33.817, -56.245, 91.311, -129.823, 46.426, 141.259]
  MoveL 3805 to (329.14, -6, -316.14) mm, rotated rx -179.9 ry 0 rz -90 deg; joints [33.827, -56.246, 91.313, -129.813, 46.433, 141.252]
  MoveL 3806 to (329.35, -6, -315.96) mm, rotated rx -179.9 ry 0 rz -90 deg; joints [33.837, -56.248, 91.317, -129.803, 46.44, 141.246]
  MoveL 3807 to (329.58, -6, -315.74) mm, rotated rx -179.9 ry 0 rz -90 deg; joints [33.849, -56.251, 91.322, -129.792, 46.448, 141.239]
  MoveL 3808 to (329.82, -6, -315.49) mm, rotated rx -179.9 ry 0 rz -90 deg; joints [33.861, -56.256, 91.329, -129.781, 46.457, 141.233]
  MoveL 3809 to (330, -6, -315.27) mm, rotated rx -179.9 ry 0 rz -90 deg; joints [33.871, -56.261, 91.336, -129.772, 46.465, 141.229]
  MoveL 3810 to (330.17, -6, -315.06) mm, rotated rx -179.9 ry 0 rz -90 deg; joints [33.88, -56.266, 91.345, -129.764, 46.473, 141.225]
  MoveL 3811 to (330.47, -6, -314.63) mm, rotated rx -179.9 ry 0 rz -90 deg; joints [33.898, -56.278, 91.363, -129.75, 46.489, 141.22]
  MoveL 3812 to (330.72, -6, -314.2) mm, rotated rx -179.9 ry 0 rz -90 deg; joints [33.914, -56.292, 91.385, -129.739, 46.504, 141.217]
  MoveL 3813 to (330.74, -6, -314.16) mm, rotated rx -179.9 ry 0 rz -90 deg; joints [33.916, -56.293, 91.387, -129.738, 46.505, 141.216]
  MoveL 3814 to (330.95, -6, -313.71) mm, rotated rx -179.9 ry 0 rz -90 deg; joints [33.931, -56.309, 91.412, -129.728, 46.521, 141.215]
  MoveL 3815 to (331.12, -6, -313.26) mm, rotated rx -179.9 ry 0 rz -90 deg; joints [33.945, -56.326, 91.44, -129.72, 46.537, 141.216]
  MoveL 3816 to (331.26, -6, -312.81) mm, rotated rx -179.9 ry 0 rz -90 deg; joints [33.959, -56.345, 91.469, -129.714, 46.552, 141.218]
  MoveL 3817 to (331.35, -6, -312.37) mm, rotated rx -179.9 ry 0 rz -90 deg; joints [33.971, -56.365, 91.501, -129.71, 46.567, 141.222]
  MoveL 3818 to (331.42, -6, -311.92) mm, rotated rx -179.9 ry 0 rz -90 deg; joints [33.982, -56.386, 91.534, -129.707, 46.582, 141.227]
  MoveL 3819 to (331.45, -6, -311.47) mm, rotated rx -179.9 ry 0 rz -90 deg; joints [33.992, -56.408, 91.57, -129.706, 46.597, 141.234]
  MoveL 3820 to (331.45, -6, -310.57) mm, rotated rx -179.9 ry 0 rz -90 deg; joints [34.01, -56.454, 91.643, -129.706, 46.626, 141.25]
  MoveL 3821 to (331.45, -6, -3.46) mm, rotated rx -179.9 ry 0 rz -90 deg; joints [41.446, -71.038, 113.329, -126.647, 55.571, 143.8]
  MoveL 3822 to (331.45, -6, -2.56) mm, rotated rx -179.9 ry 0 rz -90 deg; joints [41.472, -71.078, 113.384, -126.63, 55.594, 143.8]
  MoveL 3823 to (331.42, -6, -2.11) mm, rotated rx -179.9 ry 0 rz -90 deg; joints [41.484, -71.1, 113.412, -126.622, 55.606, 143.801]
  MoveL 3824 to (331.36, -6, -1.67) mm, rotated rx -179.9 ry 0 rz -90 deg; joints [41.495, -71.122, 113.443, -126.616, 55.617, 143.804]
  MoveL 3825 to (331.27, -6, -1.22) mm, rotated rx -179.9 ry 0 rz -90 deg; joints [41.504, -71.145, 113.475, -126.611, 55.628, 143.807]
  MoveL 3826 to (331.14, -6, -0.77) mm, rotated rx -179.9 ry 0 rz -90 deg; joints [41.513, -71.17, 113.509, -126.608, 55.639, 143.811]
  MoveL 3827 to (330.97, -6, -0.32) mm, rotated rx -179.9 ry 0 rz -90 deg; joints [41.521, -71.197, 113.545, -126.606, 55.649, 143.816]
  MoveL 3828 to (330.77, -6, 0.13) mm, rotated rx -179.9 ry 0 rz -90 deg; joints [41.527, -71.225, 113.584, -126.605, 55.659, 143.823]
  MoveL 3829 to (330.72, -6, 0.23) mm, rotated rx -179.9 ry 0 rz -90 deg; joints [41.528, -71.231, 113.592, -126.606, 55.661, 143.825]
  MoveL 3830 to (330.49, -6, 0.63) mm, rotated rx -179.9 ry 0 rz -90 deg; joints [41.532, -71.258, 113.629, -126.607, 55.669, 143.832]
  MoveL 3831 to (330.21, -6, 1.03) mm, rotated rx -179.9 ry 0 rz -90 deg; joints [41.535, -71.286, 113.668, -126.61, 55.677, 143.841]
  MoveL 3832 to (330.03, -6, 1.27) mm, rotated rx -179.9 ry 0 rz -90 deg; joints [41.535, -71.304, 113.692, -126.613, 55.682, 143.847]
  MoveL 3833 to (329.82, -6, 1.51) mm, rotated rx -179.9 ry 0 rz -90 deg; joints [41.536, -71.323, 113.718, -126.617, 55.686, 143.854]
  MoveL 3834 to (329.62, -6, 1.72) mm, rotated rx -179.9 ry 0 rz -90 deg; joints [41.535, -71.34, 113.741, -126.62, 55.69, 143.86]
  MoveL 3835 to (329.41, -6, 1.93) mm, rotated rx -179.9 ry 0 rz -90 deg; joints [41.534, -71.357, 113.765, -126.625, 55.693, 143.867]
  MoveL 3836 to (329.16, -6, 2.14) mm, rotated rx -179.9 ry 0 rz -90 deg; joints [41.533, -71.376, 113.791, -126.631, 55.696, 143.875]
  MoveL 3837 to (328.92, -6, 2.33) mm, rotated rx -179.9 ry 0 rz -90 deg; joints [41.53, -71.394, 113.816, -126.637, 55.699, 143.883]
  MoveL 3838 to (328.54, -6, 2.6) mm, rotated rx -179.9 ry 0 rz -90 deg; joints [41.526, -71.421, 113.853, -126.647, 55.702, 143.895]
  MoveL 3839 to (328.16, -6, 2.82) mm, rotated rx -179.9 ry 0 rz -90 deg; joints [41.52, -71.446, 113.887, -126.657, 55.704, 143.907]
  MoveL 3840 to (328.02, -6, 2.9) mm, rotated rx -179.9 ry 0 rz -90 deg; joints [41.517, -71.454, 113.899, -126.661, 55.705, 143.912]
  MoveL 3841 to (327.57, -6, 3.11) mm, rotated rx -179.9 ry 0 rz -90 deg; joints [41.509, -71.481, 113.936, -126.675, 55.706, 143.926]
  MoveL 3842 to (327.12, -6, 3.28) mm, rotated rx -179.9 ry 0 rz -90 deg; joints [41.499, -71.506, 113.97, -126.69, 55.706, 143.94]
  MoveL 3843 to (326.67, -6, 3.41) mm, rotated rx -179.9 ry 0 rz -90 deg; joints [41.488, -71.529, 114.002, -126.705, 55.705, 143.955]
  MoveL 3844 to (326.22, -6, 3.51) mm, rotated rx -179.9 ry 0 rz -90 deg; joints [41.477, -71.551, 114.032, -126.721, 55.703, 143.969]
  MoveL 3845 to (325.77, -6, 3.57) mm, rotated rx -179.9 ry 0 rz -90 deg; joints [41.464, -71.571, 114.06, -126.738, 55.7, 143.983]
  MoveL 3846 to (325.33, -6, 3.6) mm, rotated rx -179.9 ry 0 rz -90 deg; joints [41.45, -71.59, 114.087, -126.755, 55.696, 143.998]
  MoveL 3847 to (324.43, -6, 3.61) mm, rotated rx -179.9 ry 0 rz -90 deg; joints [41.421, -71.625, 114.135, -126.791, 55.687, 144.027]
  MoveL 3848 to (319.96, -6, 3.61) mm, rotated rx -179.9 ry 0 rz -90 deg; joints [41.276, -71.798, 114.375, -126.97, 55.642, 144.169]
  MoveL 3849 to (319.95, -6, 3.61) mm, rotated rx -179.9 ry 0 rz -90 deg; joints [41.275, -71.798, 114.376, -126.971, 55.642, 144.17]
  MoveL 3850 to (319.93, -6, 3.62) mm, rotated rx -179.9 ry 0 rz -90 deg; joints [41.275, -71.799, 114.377, -126.971, 55.642, 144.17]
  MoveL 3851 to (319.83, -6, 3.72) mm, rotated rx -179.9 ry 0 rz -90 deg; joints [41.275, -71.808, 114.389, -126.973, 55.643, 144.174]
  MoveL 3852 to (319.43, -6, 4.05) mm, rotated rx -179.9 ry 0 rz -90 deg; joints [41.271, -71.838, 114.43, -126.983, 55.648, 144.186]
  MoveL 3853 to (319.03, -6, 4.33) mm, rotated rx -179.9 ry 0 rz -90 deg; joints [41.266, -71.866, 114.468, -126.993, 55.651, 144.199]
  MoveL 3854 to (318.78, -6, 4.48) mm, rotated rx -179.9 ry 0 rz -90 deg; joints [41.263, -71.882, 114.49, -127, 55.653, 144.206]
  MoveL 3855 to (318.54, -6, 4.62) mm, rotated rx -179.9 ry 0 rz -90 deg; joints [41.258, -71.898, 114.512, -127.007, 55.654, 144.214]
  MoveL 3856 to (318.14, -6, 4.81) mm, rotated rx -179.9 ry 0 rz -90 deg; joints [41.251, -71.922, 114.545, -127.02, 55.655, 144.227]
  MoveL 3857 to (317.69, -6, 4.99) mm, rotated rx -179.9 ry 0 rz -90 deg; joints [41.241, -71.947, 114.58, -127.034, 55.655, 144.241]
  MoveL 3858 to (317.24, -6, 5.13) mm, rotated rx -179.9 ry 0 rz -90 deg; joints [41.231, -71.971, 114.612, -127.049, 55.654, 144.255]
  MoveL 3859 to (316.79, -6, 5.23) mm, rotated rx -179.9 ry 0 rz -90 deg; joints [41.219, -71.993, 114.642, -127.065, 55.652, 144.27]
  MoveL 3860 to (316.34, -6, 5.3) mm, rotated rx -179.9 ry 0 rz -90 deg; joints [41.206, -72.013, 114.67, -127.082, 55.649, 144.284]
  MoveL 3861 to (315.89, -6, 5.34) mm, rotated rx -179.9 ry 0 rz -90 deg; joints [41.193, -72.032, 114.697, -127.099, 55.645, 144.298]
  MoveL 3862 to (315.44, -6, 5.35) mm, rotated rx -179.9 ry 0 rz -90 deg; joints [41.178, -72.05, 114.721, -127.117, 55.641, 144.313]
  MoveL 3863 to (-302.86, -6, 5.35) mm, rotated rx -179.9 ry 0 rz -90 deg; joints [14.006, -90.246, 136.56, -160.686, 47.012, 167.005]
  MoveL 3864 to (-303.31, -6, 5.35) mm, rotated rx -179.9 ry 0 rz -90 deg; joints [13.982, -90.253, 136.567, -160.719, 47.006, 167.027]
  MoveL 3865 to (-303.76, -6, 5.31) mm, rotated rx -179.9 ry 0 rz -90 deg; joints [13.957, -90.258, 136.572, -160.752, 47.001, 167.049]
  MoveL 3866 to (-304.21, -6, 5.25) mm, rotated rx -179.9 ry 0 rz -90 deg; joints [13.931, -90.261, 136.576, -160.786, 46.995, 167.072]
  MoveL 3867 to (-304.66, -6, 5.15) mm, rotated rx -179.9 ry 0 rz -90 deg; joints [13.905, -90.262, 136.577, -160.82, 46.989, 167.095]
  MoveL 3868 to (-305.1, -6, 5.01) mm, rotated rx -179.9 ry 0 rz -90 deg; joints [13.879, -90.26, 136.575, -160.856, 46.984, 167.119]
  MoveL 3869 to (-305.55, -6, 4.84) mm, rotated rx -179.9 ry 0 rz -90 deg; joints [13.852, -90.256, 136.571, -160.892, 46.978, 167.143]
  MoveL 3870 to (-306.02, -6, 4.62) mm, rotated rx -179.9 ry 0 rz -90 deg; joints [13.824, -90.249, 136.565, -160.929, 46.972, 167.169]
  MoveL 3871 to (-306.45, -6, 4.37) mm, rotated rx -179.9 ry 0 rz -90 deg; joints [13.797, -90.239, 136.556, -160.966, 46.966, 167.193]
  MoveL 3872 to (-306.88, -6, 4.07) mm, rotated rx -179.9 ry 0 rz -90 deg; joints [13.769, -90.226, 136.543, -161.002, 46.961, 167.218]
  MoveL 3873 to (-307.31, -6, 3.72) mm, rotated rx -179.9 ry 0 rz -90 deg; joints [13.741, -90.21, 136.528, -161.04, 46.955, 167.243]
  MoveL 3874 to (-307.35, -6, 3.68) mm, rotated rx -179.9 ry 0 rz -90 deg; joints [13.738, -90.208, 136.526, -161.044, 46.955, 167.246]
  MoveL 3875 to (-307.41, -6, 3.63) mm, rotated rx -179.9 ry 0 rz -90 deg; joints [13.735, -90.205, 136.523, -161.049, 46.954, 167.249]
  MoveL 3876 to (-307.42, -6, 3.62) mm, rotated rx -179.9 ry 0 rz -90 deg; joints [13.734, -90.205, 136.523, -161.05, 46.954, 167.25]
  MoveL 3877 to (-307.44, -6, 3.61) mm, rotated rx -179.9 ry 0 rz -90 deg; joints [13.733, -90.204, 136.522, -161.052, 46.953, 167.251]
  MoveL 3878 to (-319.03, -6, 3.61) mm, rotated rx -179.9 ry 0 rz -90 deg; joints [13.097, -90.385, 136.706, -161.902, 46.816, 167.822]
  MoveL 3879 to (-319.93, -6, 3.6) mm, rotated rx -179.9 ry 0 rz -90 deg; joints [13.048, -90.399, 136.719, -161.968, 46.806, 167.867]
  MoveL 3880 to (-320.38, -6, 3.56) mm, rotated rx -179.9 ry 0 rz -90 deg; joints [13.023, -90.403, 136.723, -162.002, 46.801, 167.89]
  MoveL 3881 to (-320.83, -6, 3.48) mm, rotated rx -179.9 ry 0 rz -90 deg; joints [12.997, -90.405, 136.726, -162.036, 46.795, 167.913]
  MoveL 3882 to (-321.28, -6, 3.38) mm, rotated rx -179.9 ry 0 rz -90 deg; joints [12.971, -90.404, 136.726, -162.071, 46.79, 167.936]
  MoveL 3883 to (-321.73, -6, 3.24) mm, rotated rx -179.9 ry 0 rz -90 deg; joints [12.944, -90.402, 136.723, -162.107, 46.785, 167.96]
  MoveL 3884 to (-321.8, -6, 3.21) mm, rotated rx -179.9 ry 0 rz -90 deg; joints [12.94, -90.401, 136.723, -162.113, 46.784, 167.964]
  MoveC 3885 to (-322.77, -6, 3.3) mm, rotated rx -179.9 ry 0 rz -90 deg; joints [12.888, -90.422, 136.743, -162.183, 46.773, 168.012] to (-323.4, -6, 4.04) mm, rotated rx -179.9 ry 0 rz -90 deg; joints [12.863, -90.481, 136.801, -162.216, 46.766, 168.033]
  MoveL 3886 to (-323.4, -6, 4.04) mm, rotated rx -179.9 ry 0 rz -90 deg; joints [12.863, -90.481, 136.801, -162.216, 46.766, 168.033]
  MoveC 3887 to (-324.26, -6, 4.88) mm, rotated rx -179.9 ry 0 rz -90 deg; joints [12.826, -90.55, 136.868, -162.264, 46.757, 168.066] to (-325.43, -6, 4.63) mm, rotated rx -179.9 ry 0 rz -90 deg; joints [12.758, -90.551, 136.87, -162.356, 46.743, 168.127]
  MoveL 3888 to (-325.43, -6, 4.63) mm, rotated rx -179.9 ry 0 rz -90 deg; joints [12.758, -90.55, 136.87, -162.356, 46.743, 168.127]
  MoveC 3889 to (-326.15, -6, 4.33) mm, rotated rx -179.9 ry 0 rz -90 deg; joints [12.715, -90.541, 136.861, -162.414, 46.735, 168.167] to (-326.9, -6, 4.51) mm, rotated rx -179.9 ry 0 rz -90 deg; joints [12.676, -90.564, 136.884, -162.467, 46.727, 168.202]
  MoveL 3890 to (-326.9, -6, 4.51) mm, rotated rx -179.9 ry 0 rz -90 deg; joints [12.676, -90.564, 136.884, -162.467, 46.727, 168.202]
  MoveC 3891 to (-328.97, -6, 12.79) mm, rotated rx -179.9 ry 0 rz -90 deg; joints [12.665, -91.152, 137.45, -162.475, 46.703, 168.203] to (-320.69, -6, 14.85) mm, rotated rx -179.9 ry 0 rz -90 deg; joints [13.152, -91.166, 137.458, -161.82, 46.801, 167.761]
  MoveL 3892 to (-320.69, -6, 14.85) mm, rotated rx -179.9 ry 0 rz -90 deg; joints [13.152, -91.166, 137.458, -161.82, 46.801, 167.761]
  MoveC 3893 to (-318.2, -6, 7.43) mm, rotated rx -179.9 ry 0 rz -90 deg; joints [13.193, -90.628, 136.94, -161.772, 46.829, 167.733] to (-325.14, -6, 3.8) mm, rotated rx -179.9 ry 0 rz -90 deg; joints [12.764, -90.491, 136.812, -162.349, 46.746, 168.123]
  MoveL 3894 to (-325.14, -6, 3.8) mm, rotated rx -179.9 ry 0 rz -90 deg; joints [12.764, -90.491, 136.812, -162.349, 46.746, 168.123]
  MoveL 3895 to (-325.19, -6, 3.81) mm, rotated rx -179.9 ry 0 rz -90 deg; joints [12.761, -90.492, 136.813, -162.352, 46.746, 168.125]
  MoveL 3896 to (-327.18, -6.08, 4.69) mm, rotated rx -179.9 ry 0 rz -90 deg; joints [12.662, -90.577, 136.903, -162.487, 46.73, 168.217]
  MoveL 3897 to (-328.74, -6.15, 6.22) mm, rotated rx -179.9 ry 0 rz -90 deg; joints [12.596, -90.699, 137.028, -162.577, 46.719, 168.279]
  MoveL 3898 to (-329.65, -6.23, 8.21) mm, rotated rx -179.9 ry 0 rz -90 deg; joints [12.57, -90.842, 137.173, -162.612, 46.715, 168.302]
  MoveL 3899 to (-329.79, -6.31, 10.39) mm, rotated rx -179.9 ry 0 rz -90 deg; joints [12.589, -90.987, 137.319, -162.586, 46.72, 168.285]
  MoveL 3900 to (-329.15, -6.38, 12.47) mm, rotated rx -179.9 ry 0 rz -90 deg; joints [12.651, -91.114, 137.446, -162.503, 46.733, 168.229]
  MoveL 3901 to (-327.8, -6.46, 14.19) mm, rotated rx -179.9 ry 0 rz -90 deg; joints [12.748, -91.207, 137.54, -162.374, 46.755, 168.143]
  MoveL 3902 to (-325.94, -6.54, 15.32) mm, rotated rx -179.9 ry 0 rz -90 deg; joints [12.866, -91.251, 137.588, -162.216, 46.782, 168.037]
  MoveL 3903 to (-323.79, -6.61, 15.72) mm, rotated rx -179.9 ry 0 rz -90 deg; joints [12.991, -91.241, 137.583, -162.05, 46.814, 167.927]
  MoveL 3904 to (-321.64, -6.69, 15.32) mm, rotated rx -179.9 ry 0 rz -90 deg; joints [13.105, -91.178, 137.528, -161.9, 46.846, 167.828]
  MoveL 3905 to (-319.78, -6.77, 14.18) mm, rotated rx -179.9 ry 0 rz -90 deg; joints [13.194, -91.069, 137.429, -161.784, 46.875, 167.753]
  MoveL 3906 to (-318.44, -6.84, 12.46) mm, rotated rx -179.9 ry 0 rz -90 deg; joints [13.245, -90.928, 137.3, -161.718, 46.897, 167.711]
  MoveL 3907 to (-317.8, -6.92, 10.37) mm, rotated rx -179.9 ry 0 rz -90 deg; joints [13.253, -90.774, 137.158, -161.711, 46.911, 167.709]
  MoveL 3908 to (-317.95, -7, 8.2) mm, rotated rx -179.9 ry 0 rz -90 deg; joints [13.217, -90.627, 137.023, -161.764, 46.914, 167.747]
  MoveL 3909 to (-318.86, -7.07, 6.21) mm, rotated rx -179.9 ry 0 rz -90 deg; joints [13.141, -90.505, 136.912, -161.868, 46.908, 167.82]
  MoveL 3910 to (-320.42, -7.15, 4.68) mm, rotated rx -179.9 ry 0 rz -90 deg; joints [13.035, -90.422, 136.84, -162.012, 46.895, 167.919]
  MoveL 3911 to (-322.42, -7.23, 3.81) mm, rotated rx -179.9 ry 0 rz -90 deg; joints [12.914, -90.391, 136.816, -162.177, 46.878, 168.031]
  MoveL 3912 to (-324.6, -7.3, 3.7) mm, rotated rx -179.9 ry 0 rz -90 deg; joints [12.793, -90.412, 136.845, -162.342, 46.859, 168.143]
  MoveL 3913 to (-326.67, -7.38, 4.38) mm, rotated rx -179.9 ry 0 rz -90 deg; joints [12.687, -90.485, 136.923, -162.485, 46.842, 168.241]
  MoveL 3914 to (-328.37, -7.46, 5.75) mm, rotated rx -179.9 ry 0 rz -90 deg; joints [12.61, -90.598, 137.04, -162.589, 46.83, 168.312]
  MoveL 3915 to (-329.47, -7.53, 7.63) mm, rotated rx -179.9 ry 0 rz -90 deg; joints [12.573, -90.737, 137.182, -162.64, 46.825, 168.346]
  MoveL 3916 to (-329.83, -7.61, 9.79) mm, rotated rx -179.9 ry 0 rz -90 deg; joints [12.58, -90.883, 137.329, -162.63, 46.827, 168.34]
  MoveL 3917 to (-329.4, -7.69, 11.93) mm, rotated rx -179.9 ry 0 rz -90 deg; joints [12.631, -91.017, 137.464, -162.562, 46.838, 168.295]
  MoveL 3918 to (-328.23, -7.76, 13.77) mm, rotated rx -179.9 ry 0 rz -90 deg; joints [12.719, -91.121, 137.568, -162.445, 46.857, 168.216]
  MoveL 3919 to (-326.49, -7.84, 15.08) mm, rotated rx -179.9 ry 0 rz -90 deg; joints [12.833, -91.179, 137.629, -162.293, 46.884, 168.115]
  MoveL 3920 to (-324.39, -7.92, 15.69) mm, rotated rx -179.9 ry 0 rz -90 deg; joints [12.958, -91.184, 137.639, -162.127, 46.915, 168.005]
  MoveL 3921 to (-322.21, -7.99, 15.5) mm, rotated rx -179.9 ry 0 rz -90 deg; joints [13.076, -91.135, 137.597, -161.971, 46.947, 167.901]
  MoveL 3922 to (-320.25, -8.07, 14.56) mm, rotated rx -179.9 ry 0 rz -90 deg; joints [13.173, -91.037, 137.509, -161.844, 46.977, 167.819]
  MoveL 3923 to (-318.74, -8.15, 12.98) mm, rotated rx -179.9 ry 0 rz -90 deg; joints [13.236, -90.903, 137.387, -161.764, 47.001, 167.767]
  MoveL 3924 to (-317.9, -8.22, 10.96) mm, rotated rx -179.9 ry 0 rz -90 deg; joints [13.256, -90.751, 137.247, -161.74, 47.017, 167.754]
  MoveL 3925 to (-317.83, -8.3, 8.78) mm, rotated rx -179.9 ry 0 rz -90 deg; joints [13.232, -90.6, 137.107, -161.776, 47.022, 167.781]
  MoveL 3926 to (-318.54, -8.38, 6.72) mm, rotated rx -179.9 ry 0 rz -90 deg; joints [13.166, -90.47, 136.988, -161.868, 47.019, 167.845]
  MoveL 3927 to (-319.94, -8.45, 5.04) mm, rotated rx -179.9 ry 0 rz -90 deg; joints [13.067, -90.375, 136.904, -162.002, 47.008, 167.938]
  MoveL 3928 to (-321.84, -8.53, 3.98) mm, rotated rx -179.9 ry 0 rz -90 deg; joints [12.949, -90.329, 136.866, -162.163, 46.991, 168.047]
  MoveL 3929 to (-324, -8.61, 3.65) mm, rotated rx -179.9 ry 0 rz -90 deg; joints [12.826, -90.336, 136.881, -162.329, 46.973, 168.161]
  MoveL 3930 to (-326.13, -8.68, 4.12) mm, rotated rx -179.9 ry 0 rz -90 deg; joints [12.714, -90.395, 136.947, -162.48, 46.955, 168.263]
  MoveL 3931 to (-327.96, -8.76, 5.32) mm, rotated rx -179.9 ry 0 rz -90 deg; joints [12.628, -90.499, 137.054, -162.597, 46.942, 168.342]
  MoveL 3932 to (-329.24, -8.83, 7.08) mm, rotated rx -179.9 ry 0 rz -90 deg; joints [12.58, -90.632, 137.191, -162.663, 46.934, 168.387]
  MoveL 3933 to (-329.81, -8.91, 9.19) mm, rotated rx -179.9 ry 0 rz -90 deg; joints [12.574, -90.778, 137.338, -162.67, 46.935, 168.392]
  MoveL 3934 to (-329.59, -8.99, 11.36) mm, rotated rx -179.9 ry 0 rz -90 deg; joints [12.614, -90.918, 137.478, -162.618, 46.944, 168.357]
  MoveL 3935 to (-328.62, -9.06, 13.31) mm, rotated rx -179.9 ry 0 rz -90 deg; joints [12.692, -91.031, 137.593, -162.513, 46.961, 168.287]
  MoveL 3936 to (-327.01, -9.14, 14.79) mm, rotated rx -179.9 ry 0 rz -90 deg; joints [12.801, -91.103, 137.667, -162.368, 46.986, 168.191]
  MoveL 3937 to (-324.98, -9.22, 15.6) mm, rotated rx -179.9 ry 0 rz -90 deg; joints [12.924, -91.123, 137.691, -162.205, 47.015, 168.082]
  MoveL 3938 to (-322.8, -9.29, 15.63) mm, rotated rx -179.9 ry 0 rz -90 deg; joints [13.046, -91.088, 137.663, -162.044, 47.048, 167.976]
  MoveL 3939 to (-320.75, -9.37, 14.89) mm, rotated rx -179.9 ry 0 rz -90 deg; joints [13.15, -91.002, 137.586, -161.907, 47.078, 167.887]
  MoveL 3940 to (-319.1, -9.45, 13.46) mm, rotated rx -179.9 ry 0 rz -90 deg; joints [13.223, -90.877, 137.472, -161.813, 47.104, 167.826]
  MoveL 3941 to (-318.06, -9.52, 11.54) mm, rotated rx -179.9 ry 0 rz -90 deg; joints [13.256, -90.728, 137.335, -161.773, 47.122, 167.802]
  MoveL 3942 to (-318.04, -9.53, 11.5) mm, rotated rx -179.9 ry 0 rz -90 deg; joints [13.256, -90.725, 137.332, -161.773, 47.122, 167.802]
  MoveL 3943 to (-317.84, -9.53, 10.85) mm, rotated rx -179.9 ry 0 rz -90 deg; joints [13.259, -90.678, 137.286, -161.77, 47.124, 167.8]
  MoveC 3944 to (-318.24, -9.53, 6.21) mm, rotated rx -179.9 ry 0 rz -90 deg; joints [13.176, -90.374, 136.992, -161.883, 47.116, 167.878] to (-321.8, -9.53, 3.21) mm, rotated rx -179.9 ry 0 rz -90 deg; joints [12.941, -90.229, 136.853, -162.197, 47.072, 168.09]
  MoveL 3945 to (-321.8, -9.53, 3.21) mm, rotated rx -179.9 ry 0 rz -90 deg; joints [12.941, -90.229, 136.853, -162.197, 47.072, 168.09]
  MoveL 3946 to (-326.22, -9.53, 1.82) mm, rotated rx -179.9 ry 0 rz -90 deg; joints [12.681, -90.202, 136.829, -162.547, 47.022, 168.325]
  MoveL 3947 to (-327.12, -9.53, 1.53) mm, rotated rx -179.9 ry 0 rz -90 deg; joints [12.628, -90.196, 136.824, -162.618, 47.011, 168.372]
  MoveL 3948 to (-327.35, -9.52, 1.45) mm, rotated rx -179.9 ry 0 rz -90 deg; joints [12.614, -90.194, 136.822, -162.636, 47.009, 168.384]
  MoveL 3949 to (-327.57, -9.53, 1.36) mm, rotated rx -179.9 ry 0 rz -90 deg; joints [12.601, -90.191, 136.82, -162.654, 47.006, 168.397]
  MoveL 3950 to (-327.8, -9.53, 1.26) mm, rotated rx -179.9 ry 0 rz -90 deg; joints [12.587, -90.188, 136.817, -162.672, 47.004, 168.409]
  MoveL 3951 to (-328.02, -9.53, 1.15) mm, rotated rx -179.9 ry 0 rz -90 deg; joints [12.574, -90.183, 136.813, -162.691, 47.001, 168.421]
  MoveL 3952 to (-328.25, -9.52, 1.03) mm, rotated rx -179.9 ry 0 rz -90 deg; joints [12.56, -90.179, 136.808, -162.709, 46.998, 168.434]
  MoveL 3953 to (-328.58, -9.52, 0.82) mm, rotated rx -179.9 ry 0 rz -90 deg; joints [12.539, -90.17, 136.8, -162.738, 46.995, 168.453]
  MoveL 3954 to (-328.92, -9.52, 0.58) mm, rotated rx -179.9 ry 0 rz -90 deg; joints [12.517, -90.159, 136.789, -162.766, 46.991, 168.472]
  MoveL 3955 to (-329.19, -9.53, 0.37) mm, rotated rx -179.9 ry 0 rz -90 deg; joints [12.5, -90.148, 136.779, -162.79, 46.987, 168.488]
  MoveL 3956 to (-329.46, -9.52, 0.13) mm, rotated rx -179.9 ry 0 rz -90 deg; joints [12.482, -90.136, 136.768, -162.814, 46.984, 168.504]
  MoveL 3957 to (-329.65, -9.52, -0.05) mm, rotated rx -179.9 ry 0 rz -90 deg; joints [12.469, -90.127, 136.759, -162.831, 46.982, 168.516]
  MoveL 3958 to (-329.82, -9.52, -0.24) mm, rotated rx -179.9 ry 0 rz -90 deg; joints [12.458, -90.117, 136.749, -162.847, 46.98, 168.526]
  MoveL 3959 to (-330.04, -9.53, -0.5) mm, rotated rx -179.9 ry 0 rz -90 deg; joints [12.442, -90.103, 136.735, -162.868, 46.977, 168.541]
  MoveL 3960 to (-330.25, -9.53, -0.77) mm, rotated rx -179.9 ry 0 rz -90 deg; joints [12.428, -90.088, 136.721, -162.887, 46.975, 168.554]
  MoveL 3961 to (-330.5, -9.53, -1.15) mm, rotated rx -179.9 ry 0 rz -90 deg; joints [12.409, -90.066, 136.7, -162.912, 46.972, 168.571]
  MoveL 3962 to (-330.72, -9.53, -1.53) mm, rotated rx -179.9 ry 0 rz -90 deg; joints [12.392, -90.044, 136.678, -162.934, 46.969, 168.586]
  MoveL 3963 to (-330.79, -9.53, -1.67) mm, rotated rx -179.9 ry 0 rz -90 deg; joints [12.387, -90.036, 136.67, -162.942, 46.968, 168.591]
  MoveL 3964 to (-330.99, -9.52, -2.11) mm, rotated rx -179.9 ry 0 rz -90 deg; joints [12.37, -90.009, 136.644, -162.964, 46.965, 168.606]
  MoveL 3965 to (-331.15, -9.53, -2.56) mm, rotated rx -179.9 ry 0 rz -90 deg; joints [12.356, -89.981, 136.617, -162.984, 46.963, 168.619]
  MoveL 3966 to (-331.28, -9.52, -3.01) mm, rotated rx -179.9 ry 0 rz -90 deg; joints [12.344, -89.953, 136.59, -163, 46.961, 168.63]
  MoveL 3967 to (-331.37, -9.52, -3.46) mm, rotated rx -179.9 ry 0 rz -90 deg; joints [12.333, -89.924, 136.562, -163.014, 46.96, 168.64]
  MoveL 3968 to (-331.42, -9.53, -3.91) mm, rotated rx -179.9 ry 0 rz -90 deg; joints [12.325, -89.895, 136.533, -163.026, 46.959, 168.648]
  MoveL 3969 to (-331.45, -9.52, -4.36) mm, rotated rx -179.9 ry 0 rz -90 deg; joints [12.318, -89.866, 136.504, -163.035, 46.958, 168.654]
  MoveL 3970 to (-331.45, -9.52, -5.26) mm, rotated rx -179.9 ry 0 rz -90 deg; joints [12.307, -89.806, 136.446, -163.05, 46.957, 168.664]
  MoveL 3971 to (-331.45, -9.53, -310.57) mm, rotated rx -179.9 ry 0 rz -90 deg; joints [9.463, -71.168, 114.407, -166.095, 43.143, 170.129]
  MoveL 3972 to (-331.44, -9.52, -311.47) mm, rotated rx -179.9 ry 0 rz -90 deg; joints [9.457, -71.116, 114.335, -166.099, 43.123, 170.128]
  MoveL 3973 to (-331.41, -9.53, -311.92) mm, rotated rx -179.9 ry 0 rz -90 deg; joints [9.455, -71.09, 114.299, -166.099, 43.113, 170.127]
  MoveL 3974 to (-331.35, -9.52, -312.37) mm, rotated rx -179.9 ry 0 rz -90 deg; joints [9.454, -71.063, 114.263, -166.098, 43.104, 170.124]
  MoveL 3975 to (-331.25, -9.53, -312.81) mm, rotated rx -179.9 ry 0 rz -90 deg; joints [9.455, -71.036, 114.225, -166.094, 43.094, 170.119]
  MoveL 3976 to (-331.12, -9.52, -313.26) mm, rotated rx -179.9 ry 0 rz -90 deg; joints [9.458, -71.009, 114.188, -166.087, 43.085, 170.113]
  MoveL 3977 to (-330.95, -9.53, -313.71) mm, rotated rx -179.9 ry 0 rz -90 deg; joints [9.462, -70.981, 114.15, -166.079, 43.075, 170.105]
  MoveL 3978 to (-330.73, -9.53, -314.16) mm, rotated rx -179.9 ry 0 rz -90 deg; joints [9.468, -70.953, 114.111, -166.068, 43.066, 170.095]
  MoveL 3979 to (-330.72, -9.52, -314.19) mm, rotated rx -179.9 ry 0 rz -90 deg; joints [9.468, -70.951, 114.108, -166.067, 43.065, 170.095]
  MoveL 3980 to (-330.47, -9.52, -314.63) mm, rotated rx -179.9 ry 0 rz -90 deg; joints [9.476, -70.924, 114.07, -166.053, 43.056, 170.083]
  MoveL 3981 to (-330.17, -9.52, -315.06) mm, rotated rx -179.9 ry 0 rz -90 deg; joints [9.485, -70.896, 114.032, -166.037, 43.048, 170.069]
  MoveL 3982 to (-329.82, -9.52, -315.48) mm, rotated rx -179.9 ry 0 rz -90 deg; joints [9.497, -70.868, 113.993, -166.017, 43.039, 170.053]
  MoveL 3983 to (-329.58, -9.53, -315.73) mm, rotated rx -179.9 ry 0 rz -90 deg; joints [9.505, -70.851, 113.97, -166.003, 43.035, 170.042]
  MoveL 3984 to (-329.34, -9.52, -315.96) mm, rotated rx -179.9 ry 0 rz -90 deg; joints [9.514, -70.836, 113.949, -165.989, 43.03, 170.032]
  MoveL 3985 to (-329.13, -9.53, -316.14) mm, rotated rx -179.9 ry 0 rz -90 deg; joints [9.522, -70.823, 113.931, -165.977, 43.027, 170.022]
  MoveL 3986 to (-328.92, -9.53, -316.31) mm, rotated rx -179.9 ry 0 rz -90 deg; joints [9.53, -70.812, 113.915, -165.965, 43.024, 170.012]
  MoveL 3987 to (-328.49, -9.52, -316.61) mm, rotated rx -179.9 ry 0 rz -90 deg; joints [9.546, -70.79, 113.885, -165.939, 43.019, 169.992]
  MoveL 3988 to (-328.05, -9.53, -316.86) mm, rotated rx -179.9 ry 0 rz -90 deg; joints [9.562, -70.771, 113.859, -165.913, 43.015, 169.972]
  MoveL 3989 to (-328.02, -9.52, -316.87) mm, rotated rx -179.9 ry 0 rz -90 deg; joints [9.564, -70.77, 113.858, -165.911, 43.014, 169.971]
  MoveL 3990 to (-327.57, -9.53, -317.08) mm, rotated rx -179.9 ry 0 rz -90 deg; joints [9.581, -70.754, 113.834, -165.884, 43.011, 169.95]
  MoveL 3991 to (-327.12, -9.52, -317.25) mm, rotated rx -179.9 ry 0 rz -90 deg; joints [9.599, -70.739, 113.815, -165.857, 43.009, 169.93]
  MoveL 3992 to (-326.67, -9.53, -317.39) mm, rotated rx -179.9 ry 0 rz -90 deg; joints [9.617, -70.727, 113.798, -165.829, 43.008, 169.909]
  MoveL 3993 to (-326.22, -9.52, -317.48) mm, rotated rx -179.9 ry 0 rz -90 deg; joints [9.636, -70.717, 113.784, -165.802, 43.007, 169.889]
  MoveL 3994 to (-325.77, -9.52, -317.55) mm, rotated rx -179.9 ry 0 rz -90 deg; joints [9.654, -70.709, 113.772, -165.774, 43.007, 169.868]
  MoveL 3995 to (-325.33, -9.52, -317.58) mm, rotated rx -179.9 ry 0 rz -90 deg; joints [9.673, -70.703, 113.764, -165.746, 43.008, 169.848]
  MoveL 3996 to (-324.43, -9.52, -317.59) mm, rotated rx -179.9 ry 0 rz -90 deg; joints [9.711, -70.694, 113.751, -165.69, 43.011, 169.807]
  MoveL 3997 to (324.43, -9.52, -317.59) mm, rotated rx -179.9 ry 0 rz -90 deg; joints [33.657, -56.233, 91.563, -130.187, 46.495, 141.653]
  MoveL 3998 to (325.33, -9.53, -317.58) mm, rotated rx -179.9 ry 0 rz -90 deg; joints [33.684, -56.202, 91.513, -130.144, 46.5, 141.613]
  MoveL 3999 to (325.77, -9.53, -317.55) mm, rotated rx -179.9 ry 0 rz -90 deg; joints [33.699, -56.189, 91.491, -130.122, 46.503, 141.593]
  MoveL 4000 to (326.22, -9.53, -317.49) mm, rotated rx -179.9 ry 0 rz -90 deg; joints [33.714, -56.177, 91.471, -130.1, 46.507, 141.574]
  MoveL 4001 to (326.67, -9.53, -317.39) mm, rotated rx -179.9 ry 0 rz -90 deg; joints [33.729, -56.166, 91.454, -130.079, 46.513, 141.556]
  MoveL 4002 to (327.12, -9.53, -317.26) mm, rotated rx -179.9 ry 0 rz -90 deg; joints [33.745, -56.158, 91.44, -130.057, 46.519, 141.538]
